(* CODESYS project plc_chalet_xplanar.library
   Title: CHALET_XPlanar
   Version: 5.1.2
   Placeholder: CHALET_XPlanar
   Company: Beckhoff CH

Project tree, tasks and I/O mapping:
  libraries: CHALET_BaseComponents, * (Beckhoff CH); CHALET_Nc, * (Beckhoff CH); Tc2_EtherCAT, * (Beckhoff Automation GmbH); Tc2_Math, * (Beckhoff Automation GmbH); Tc2_Standard, * (Beckhoff Automation GmbH); Tc2_System, * (Beckhoff Automation GmbH); Tc2_Utilities, * (Beckhoff Automation GmbH); Tc3_EventLogger, * (Beckhoff Automation GmbH); Tc3_Mc3Definitions, * (Beckhoff Automation GmbH); Tc3_Mc3PlanarMotion, * (Beckhoff Automation GmbH); Tc3_Module, * (Beckhoff Automation GmbH); Tc3_Physics, * (Beckhoff Automation GmbH); Tc3_XPlanarUtility, * (Beckhoff Automation GmbH)
  COMPONENTs/
    Environment/
      function block FB_XP_Environment [ST]: CollisionCheck, CollisionDetectionAlgorithm, MoverCollisionOffsetError, MoverCollisionOffsetWarning, UpdateCollisionDetection, AddToGroup, RemoveFromGroup, Clear, Configure, FB_init, Feedback, Initialize, Mapped, OID, PlanarEnvironment, Prepare, ProcessingUnitMoverDetectionStatus, ProcessingUnitOID, Update, UtilityEnvirement
      interface I_XP_Enviroment_PLC: CollisionCheck, MoverCollisionOffsetError, MoverCollisionOffsetWarning, MoverDetectionStatus, ProcessingUnitOID
      interface I_XP_Environment: AddToGroup, Clear, Configure, Feedback, Initialize, Mapped, OID, PlanarEnvironment, ProcessingUnitMoverDetectionStatus, ProcessingUnitOID, RemoveFromGroup, Update, UtilityEnvirement
    Feedback/
      function block FB_XP_Feedback [ST]: ClearObjectInfo, ObjectInfo, ObjectInfoEx
      interface I_XP_Feedback: ObjectInfo, ObjectInfoEx
      data type ST_PlanarObjectInfoEx
    Group/
      function block FB_XP_Group [ST]: AddEnvironment, AddMover, AddTrack, Disable, Enable, FB_init, Feedback, Initialize, Mapped, OID, PlanarGroup, Reset, Update
      interface I_XP_Group: AddEnvironment, AddMover, AddTrack, Disable, Enable, Feedback, Initialize, Mapped, OID, PlanarGroup, Reset, Update
    Mover/
      ProductData/
        function block FB_XP_ProductData [ST]: LinkedMover, LinkToMover
        interface I_XP_ProductData: LinkedMover, LinkToMover
      function block FB_XP_Mover [ST]: DynConstraint, SetDynConstraint_A, SetDynConstraint_B, SetDynConstraint_C, SetDynConstraint_Path, SetDynConstraint_X, SetDynConstraint_Y, SetDynConstraint_Z, AddMoverExtSetpoint, AxisExtSetpointA, AxisExtSetpointB, AxisExtSetpointC, AxisExtSetpointX, AxisExtSetpointY, AxisExtSetpointZ, StartExternalSetpoint, StopExternalSetpoint, UpdateExternalSetpoint, AddToGroup, RemoveFromGroup, Halt, MoveA, MoveB, MoveC, MoveXY, MoveZ, Standstill, Disable, Enable, Reset, LastCmdTargedGap, LastCmdTargedPosition, LastCmdTargedTrack, LastValidPositionOnTrack, LastValidPositionXYZABC, LastValidTrack, AccelerationSet, CAxisModulo, CommandMode, DistToParentStation, Enabled, LagDistanceXY, Mapped, Mode, MoverHeight, MoverIsNotPresent, MoverWidth, PositionAct, PositionSet, ProductData, Route, VelocitySet, CurrentTrack, DistToTrack, JoinTrack, MoveOnTrack, MoveOnTrack_ShortestWay, MoveOnTrackToStation, ParentStation, PositionOnTrack, TargetStation, TcIoXPlanarMover, UtilityMover, FB_init, Feedback, Initialize, OID, PlanarMover, Prepare, Update
      interface I_XP_Mover: DynConstraint, SetDynConstraint_A, SetDynConstraint_B, SetDynConstraint_C, SetDynConstraint_Path, SetDynConstraint_X, SetDynConstraint_Y, SetDynConstraint_Z, StopExternalSetpoint, AddToGroup, RemoveFromGroup, Halt, MoveA, MoveB, MoveC, MoveXY, MoveZ, Standstill, Disable, Enable, Reset, LastCmdTargedGap, LastCmdTargedPosition, LastCmdTargedTrack, LastValidPositionOnTrack, LastValidPositionXYZABC, LastValidTrack, AccelerationSet, CAxisModulo, DistToParentStation, Enabled, Feedback, Mapped, Mode, MoverHeight, MoverIsNotPresent, MoverWidth, OID, PositionSet, Route, VelocitySet, CurrentTrack, DistToTrack, JoinTrack, MoveOnTrack, MoveOnTrack_ShortestWay, MoveOnTrackToStation, ParentStation, PositionOnTrack, TargetStation, TcIoXPlanarMover, UtilityMover, PlanarMover
      interface I_XP_Mover_PLC: DynConstraint, SetDynConstraint_A, SetDynConstraint_B, SetDynConstraint_C, SetDynConstraint_Path, SetDynConstraint_X, SetDynConstraint_Y, SetDynConstraint_Z, AxisExtSetpointA, AxisExtSetpointB, AxisExtSetpointC, AxisExtSetpointX, AxisExtSetpointY, AxisExtSetpointZ, StartExternalSetpoint, StopExternalSetpoint, Halt, MoveA, MoveB, MoveC, MoveXY, MoveZ, Standstill, AccelerationSet, CAxisModulo, CommandMode, Enabled, LagDistanceXY, MoverHeight, MoverWidth, PositionAct, PositionSet, VelocitySet, CurrentTrack, LastCmdTargedGap, LastCmdTargedPosition, LastCmdTargedTrack, MoveOnTrack, ParentStation, PositionOnTrack, TargetStation, TcIoXPlanarMover, UtilityMover, DistToParentStation, Feedback, LUID, Mapped, MoverIsNotPresent, OID, PlanarMover, ProductData
    Optional/
      Casting/
        function ToXpMover [ST]
        function ToXpStation [ST]
        function ToXpTrack [ST]
      Trigger/
        function block FB_XP_Trigger [ST]: AccocietedTrack, FB_init, HR, Initialize, ListOfMoversToCheck, MoverAtTrigger, MoverDetected, PositionOnTrack, Prepare, TimeStamp, TriggerDirection, Update
        interface I_XP_Trigger: AccocietedTrack, HR, ListOfMoversToCheck, MoverAtTrigger, MoverDetected, PositionOnTrack, TimeStamp, TriggerDirection
      Zone/
        function block FB_XP_SoretedListOfMover [ST]: CtsMoversInZone, FB_init, Initialize, MoversInZone, Prepare, Update
        interface I_XP_Zone: CtsMoversInZone, MoversInZone
    Path/
      function block FB_XP_Path [ST]: DistanceToDestiantion, Length, LUID, PointerToThis, StationDestination, StationStart, TracksUsed
      interface I_XP_Path: DistanceToDestiantion, Length, PointerToThis, StationDestination, StationStart, TracksUsed
    Stationen/
      A-Star-Node/
        function block FB_AStarNode [ST]: LUID, PathLength, RouteUsedToNode, SortOrderInList, Station
        interface I_PathAStarNode: PathLength, RouteUsedToNode, Station
      function block FB_XP_Station [ST]: CheckInvalideParameter, GetAccocietedTrack, GetDecisionDistance, GetPathsAhead, GetPathsBehind, GetPosOnTrack, GetStationAhead, GetStationBehinde, SetTrackObjName, Configure, CtsEmptySpaceInQueue, CtsMoversInQueue, MoverAccAtExit, MoverDecAtExit, MoverQueueSize, MoversInPlace, MoversInQueue, MoverVelocityAtExit, OnMoverPasses, PushMoversOutOfStation, ReadyToRecvMovers, SendMoversToStation, SuppressDynamicsChange, System, TargetGroupe, TargetPosMonitoringTime, TargetPosWindow, ProcessSimulationActive, SimulationStart, SimulationStartEx, SimulationStop, UpdateSimulation, AccocietedTrack, AddMoverToQueue, AssignedMovers, DeleteMoversQueue, FB_exit, FB_init, Feedback, Filter, GetPathToTarged, Initialize, MoverGapAtExit, OID, PathsAhead, PathsBehinde, PositionOnTrack, PositionOnTrackXY, PositionXY, Prepare, StationsAhead, StationsBehinde, Update, UpdateMoverInteraction
      interface I_XP_Station: AccocietedTrack, AddMoverToQueue, AssignedMovers, Configure, CtsEmptySpaceInQueue, CtsMoversInQueue, DeleteMoversQueue, Filter, MoverAccAtExit, MoverDecAtExit, MoverGapAtExit, MoverQueueSize, MoversInPlace, MoverVelocityAtExit, PathsAhead, PathsBehinde, PositionOnTrack, PositionOnTrackXY, PositionXY, PushMoversOutOfStation, ReadyToRecvMovers, SendMoversToStation, StationsAhead, StationsBehinde, TargetGroupe, Update
      interface I_XP_Station_PLC: CtsEmptySpaceInQueue, CtsMoversInQueue, Filter, LUID, MoverAccAtExit, MoverDecAtExit, MoverQueueSize, MoversInPlace, MoversInQueue, MoverVelocityAtExit, PushMoversOutOfStation, ReadyToRecvMovers, SendMoversToStation, SuppressDynamicsChange, System, TargetPosMonitoringTime, TargetPosWindow, ProcessSimulationActive, SimulationStart, SimulationStartEx, SimulationStop, AccocietedTrack, Feedback, MoverGapAtExit, PositionOnTrack, PositionOnTrackXY, PositionXY, StationsAhead, StationsBehinde, TargetGroupe
    System/
      function block FB_XP_System [ST]: JoiningStation, JoiningTrack, Disable, Disabled, Disabling, Enable, Enabled, Enabling, FastStop, Initialize, Initialized, CheckTargetExists, GetStationClosestTo, Station, LinkEnvironment, LinkGroup, RegisterMover, RegisterStation, RegisterTrack, RegisterTrigger, RegisterZone, CheckForErrors, Enviroment, FB_init, Feedback, Movers, Paths, Stations, SuppressAllDynamicsChanges, Tracks, Triggers, Update, Zones
      interface I_XP_System_PLC: CheckTargetExists, Disable, Disabled, Enable, Enabled, Enviroment, FastStop, Feedback, GetStationClosestTo, Initialize, Initialized, Movers, Paths, Station, Stations, SuppressAllDynamicsChanges, Tracks, Triggers, Update, Zones
      interface I_XP_System_Registration: LinkEnvironment, LinkGroup, RegisterMover, RegisterStation, RegisterTrack, RegisterTrigger, RegisterZone, Disabled, Enabled, Enviroment, Movers, Paths, Stations, Tracks, Triggers, Zones
    Track/
      function block FB_XP_Track [ST]: Configure, Configuring, Disable, Enable, AddToGroup, RemoveFromGroup, AddMover, ClosedLoop, CtsMoversOnTrack, FB_init, Feedback, GapAtPosition, Initialize, Length, Mapped, MoversOnTrack, OID, PathsOnTrack, PlanarTrack, Prepare, Reset, StationAhedPosition, StationsOnTrack, TracksAhead, TracksBehinde, TracksEndAtThis, TracksStartFromThis, Update
      interface I_XP_Track: AddMover, AddToGroup, ClosedLoop, Configure, Configuring, CtsMoversOnTrack, Disable, Enable, Feedback, GapAtPosition, Length, PlanarTrack, RemoveFromGroup, Reset, StationAhedPosition, StationsOnTrack, TracksAhead, TracksBehinde, TracksEndAtThis, TracksStartFromThis
      interface I_XP_Track_PLC: CtsMoversOnTrack, Feedback, Length, Mapped, OID, PlanarTrack, StationAhedPosition, StationsOnTrack, TracksAhead, TracksBehinde, TracksEndAtThis, TracksStartFromThis
  FUNCTIONs/
    function F_DistXYVectors [ST]
    function F_Vector_Multiplication [ST]
    function F_Vector_Subtraction [ST]
    function F_GetDistToPosModulo [ST]
    function F_InLimitTest [ST]
    function F_RotatePositionXY [ST]
    function F_Vector_Addition [ST]
  00000000-0000-0000-0000-000000000000|LICENSE.md
  LICENSE.md
  global variables XPlanarParameterlist
*)

// COMPONENTs/Feedback/ST_PlanarObjectInfoEx
TYPE ST_PlanarObjectInfoEx EXTENDS Tc3_Mc3PlanarMotion.PlanarObjectInfo :
STRUCT
	ipObject : I_CH_Object;
END_STRUCT
END_TYPE

// XPlanarParameterlist
{attribute 'qualified_only'}
VAR_GLOBAL CONSTANT 
	(*After the system init, this is the first station that is approached.
	 Can be used, for example, to send all movers to the “Unload” station first 
	 The default value is “not defined” so the movers remain in the closest station and wait for a valid destination*)
	S_MOVER_TARGED_INIT : STRING := 'not defined';	
	
	(*This value as a Station.Filter allows all movers of any targed*)
	S_ANY_STATION_NAME : STRING := '';
	
	(*Only if enabled, mover take over "VelocytiAtExit" of passed station*)	
	B_STATIONS_OVERRIDE_MOVER_DYN_CONSTRAINT : BOOL := FALSE;

	(*Minimum gap center to center on track [mm] *)
	F_MOVER_MINIMUM_GAP_ON_TRACK : LREAL := 100.0;
	
	(*Default gap center to center on track. Each station can override this gap[mm] *)
	F_GAP_DEFAULT: LREAL := 120.0;
	
	(*Determine the absolute C-rotation of the mover when starting up. Requires an “APM9001-0000-4xxx | XPlanar-ID-Bumper”. *)
	B_GET_MOVER_ORIENTATION : BOOL := FALSE;	
	
	(*Add envirement to groupe during enabling *)
	B_ADD_ENVIROMENT_TO_GROUP : BOOL := TRUE;	
					
	(*Add tracks to groupe during enabling *)
	B_ADD_TRACKS_TO_GROUP : BOOL := FALSE;	
					
	(*Add movers to groupe during enabling *)
	B_ADD_MOVERS_TO_GROUP : BOOL := FALSE;	
					
	(*The movers are only sent to the next free station on the way to the destination. 
	The distance in mm can be specified here to indicate how much further away the new move command can already be sent.  *)
	F_DIST_SET_NEW_MOVE_CMD_BEFORE_REACHING_PARENT_STATION : LREAL := 200.0;
	
	(*max tracks after a track switch *)
	N_MAX_STATIONS_AHEAD_OR_BEHIND : UINT := 20;	
	
	//Velocity during enabling move on track. 0=Default
	F_ENABLING_ON_TRACK_VELOCITY	: LREAL := 0;
	
	//Acc-/Deceleration during enabling move on track. 0=Default
	F_ENABLING_ON_TRACK_ACC_DEC		: LREAL := 0;
	
	//TRUE = Use inside PLC the track name from the TcCom Track Object. If FALSE overwride TcCom Track object with instance name
	B_TRACK_NAME_TACKOVER_FROM_TRACK_OBJECT : BOOL := TRUE;
	

END_VAR

// COMPONENTs/Environment/FB_XP_Environment
{attribute 'no_explicit_call' := 'Do not call the body - Stick to OOP'}
(* XPlanar Environment - 1 per associated XPlanar 
	The Planar environment is a software object that represents the two-dimensional XPlanar stator surface. Together with Planar movers in a group, 
	it prevents collisions of the movers with the edge of the surface. *)
FUNCTION_BLOCK FB_XP_Environment EXTENDS FB_CH_Object IMPLEMENTS I_XP_Environment
VAR
	//Link to Planar-Environment object
	fbEnvironment : MC_PlanarEnvironment;
	fbUtilityEnvirement : FB_TcIoXPlanarEnvironment;
	
	{attribute 'hide'}  
	bInitDone :BOOL := FALSE;
	{attribute 'hide'}
	ipXpSystem : I_XP_System_Registration;
	{attribute 'hide'}               	
	fbFeedback 			: FB_XP_Feedback(ipSourceInfo := fbSourceInfo);	
	{attribute 'hide'}                   	
	eActiveCommand 		: CHALET_Nc.E_NcAxisCommands := CHALET_Nc.E_NcAxisCommands.None;
	{attribute 'hide'}
	bCollisionCheckEnabled : BOOL := TRUE;
	{attribute 'hide'}
	fMoverOffsetWarning : LREAL := 2.0; //[mm]
	{attribute 'hide'}
	fMoverOffsetError: LREAL := 0.0;//[mm]
	{attribute 'hide'}
	eMoverDetectionStatus : MoverDetectionStatus;
	{attribute 'hide'}
	eMoverDetectionStatusLastCycle : MoverDetectionStatus;
END_VAR


// Planar-Feedback objects
VAR
	{attribute 'hide'} 
	fbFeedbackAddToGrp : MC_PlanarFeedback;
	{attribute 'hide'} 
	fbFeedbackRmvFromGrp : MC_PlanarFeedback;
	{attribute 'hide'} 
	fbFeedbackConfigure : MC_PlanarFeedback;
	{attribute 'hide'} 
	fbFeedbackClear : MC_PlanarFeedback;
END_VAR

{attribute 'monitoring':='call'}
(* If Enable, the movers are checked for collisions with each other.
Warning and error can have their own size offsets.
The error leads to a stop with higher dynamics.
In simulation, an error does not lead to a stop *)
PROPERTY CollisionCheck : BOOL
GET
CollisionCheck := THIS^.bCollisionCheckEnabled;
END_GET
SET
THIS^.bCollisionCheckEnabled := CollisionCheck;
END_SET
END_PROPERTY

//Return an interface to the mover if a collision is active else return 0. The check stops after the first collision found
METHOD PROTECTED CollisionDetectionAlgorithm : I_XP_Mover
VAR_INPUT
	ipListOfMovers : I_CH_LIST;
	fOffsetMoverSize : LREAL := 1.0; //Offset on the mover dimension from the MC3 mover object [mm];
END_VAR
VAR
	aPointsMover1 : ARRAY[0..3] OF  Tc3_Physics.PositionXY;
	aPointsEachMover : ARRAY[0..3] OF  Tc3_Physics.PositionXY;
	aPointsDelta : ARRAY[0..3] OF  Tc3_Physics.PositionXY;
	
	fMoverWidth, fMoverHight : LREAL;
	fMoverXPos, fMoverYPos, fMoverCPos : LREAL;
	
	ipMover1, ipEachMover : I_XP_Mover;
	fbListOfMoverToCheck : FB_CH_List;
	
	fAngle : LREAL;
	a, b, c: LREAL;
	Pa, Pb, Pc : REFERENCE TO Tc3_Physics.PositionXY;
	fcos : LREAL;
	
	nIdx, nIdxMover1, nIdxPlus1 : UINT;
	ipMover2CollisionFound : I_XP_Mover;
END_VAR
//Get all mover in a list
fbListOfMoverToCheck.Duplicate(ipListOfMovers);



//Check list for invalide Act Pos - ex.: if mover is not found 
fbListOfMoverToCheck.ResetIterator();
WHILE fbListOfMoverToCheck.HasNextObject() DO
	__QUERYINTERFACE(fbListOfMoverToCheck.GetNextObject(),ipMover1);
	
	IF ipMover1.MoverIsNotPresent THEN 		
		//remove from list
		fbListOfMoverToCheck.RemoveObject(ipMover1);
		
	END_IF
END_WHILE



fbListOfMoverToCheck.ResetIterator();
WHILE fbListOfMoverToCheck.HasNextObject() DO
	//get first mover in list,
	__QUERYINTERFACE(fbListOfMoverToCheck.GetNextObject(),ipMover1);
	
	fMoverXPos := ipMover1.PlanarMover.MCTOPLC.ACT.ActPos.x;
	fMoverYPos := ipMover1.PlanarMover.MCTOPLC.ACT.ActPos.y;
	fMoverCPos := ipMover1.PlanarMover.MCTOPLC.ACT.ActPos.c;
		
	//Get corner points of the rectangle 
	fMoverWidth := ipMover1.MoverWidth - fOffsetMoverSize;
	fMoverHight := ipMover1.MoverHeight - fOffsetMoverSize;
	aPointsMover1[0].SetValuesXY(x:= -fMoverWidth/2, y:= -fMoverHight/2);//Bottom Left
	aPointsMover1[1].SetValuesXY(x:= -fMoverWidth/2, y:=  fMoverHight/2);//Top Left
	aPointsMover1[2].SetValuesXY(x:=  fMoverWidth/2, y:=  fMoverHight/2);//Top Ritgh
	aPointsMover1[3].SetValuesXY(x:=  fMoverWidth/2, y:= -fMoverHight/2);//Bottom Rigth
	
	//Rotation of the mover
	F_RotatePositionXY(aPointsMover1[0], fMoverCPos);
	F_RotatePositionXY(aPointsMover1[1], fMoverCPos);
	F_RotatePositionXY(aPointsMover1[2], fMoverCPos);
	F_RotatePositionXY(aPointsMover1[3], fMoverCPos);
	
	//shift to mover coordinates
	aPointsMover1[0].ShiftByXY(dx:= fMoverXPos, dy:= fMoverYPos);
	aPointsMover1[1].ShiftByXY(dx:= fMoverXPos, dy:= fMoverYPos);
	aPointsMover1[2].ShiftByXY(dx:= fMoverXPos, dy:= fMoverYPos);
	aPointsMover1[3].ShiftByXY(dx:= fMoverXPos, dy:= fMoverYPos);
	
	
	//do an check for all mover
	fbListOfMoverToCheck.ResetIterator();
	WHILE fbListOfMoverToCheck.HasNextObject() DO
		__QUERYINTERFACE(fbListOfMoverToCheck.GetNextObject(),ipEachMover);
		
		IF ipEachMover = ipMover1 THEN
			//Skip if same
			CONTINUE;
		END_IF
		
		fMoverXPos := ipEachMover.PlanarMover.MCTOPLC.ACT.ActPos.x;
		fMoverYPos := ipEachMover.PlanarMover.MCTOPLC.ACT.ActPos.y;
		fMovercPos := ipEachMover.PlanarMover.MCTOPLC.ACT.ActPos.c;
		
		//Get corner points of the rectangle 
		fMoverWidth := ipEachMover.MoverWidth - fOffsetMoverSize;
		fMoverHight := ipEachMover.MoverHeight - fOffsetMoverSize;
		aPointsEachMover[0].SetValuesXY(x:= -fMoverWidth/2, y:= -fMoverHight/2);//Bottom Left
		aPointsEachMover[1].SetValuesXY(x:= -fMoverWidth/2, y:=  fMoverHight/2);//Top Left
		aPointsEachMover[2].SetValuesXY(x:=  fMoverWidth/2, y:=  fMoverHight/2);//Top Ritgh
		aPointsEachMover[3].SetValuesXY(x:=  fMoverWidth/2, y:= -fMoverHight/2);//Bottom Rigth

		//Rotation of the mover
		F_RotatePositionXY(aPointsEachMover[0], fMoverCPos);
		F_RotatePositionXY(aPointsEachMover[1], fMoverCPos);
		F_RotatePositionXY(aPointsEachMover[2], fMoverCPos);
		F_RotatePositionXY(aPointsEachMover[3], fMoverCPos);
		
		//shift to mover coordinates
		aPointsEachMover[0].ShiftByXY(dx:= fMoverXPos, dy:= fMoverYPos);
		aPointsEachMover[1].ShiftByXY(dx:= fMoverXPos, dy:= fMoverYPos);
		aPointsEachMover[2].ShiftByXY(dx:= fMoverXPos, dy:= fMoverYPos);
		aPointsEachMover[3].ShiftByXY(dx:= fMoverXPos, dy:= fMoverYPos);		
		
		//check each corener if inside each mover
		FOR nIdxMover1 := 0 TO 3 DO
			
			(* A triangle is created between a corner point of Mover1 (point a) and two corner points of Mover2 (points B and C). 
			All corner points of Mover2 are now tested one after the other. If the sum of all angles "a" is 360 degrees, 
			then point A is inside mover 2 and there is a collision *)
			fAngle := 0;
			FOR nIdx := 0 TO 3 DO
				nIdxPlus1 := ((nIdx+1)MOD 4);
			
				Pa REF= aPointsMover1[nIdxMover1];
				Pb REF= aPointsEachMover[nIdx];
				Pc REF= aPointsEachMover[nIdxPlus1];					
				

				a := SQRT(EXPT((Pb.x - Pc.x),2)+EXPT((Pb.y - Pc.y),2));
				b := SQRT(EXPT((Pa.x - Pc.x),2)+EXPT((Pa.y - Pc.y),2));
				c := SQRT(EXPT((Pa.x - Pb.x),2)+EXPT((Pa.y - Pb.y),2));
				
				
				IF b=0 OR c=0 THEN
					//Error - Return the found mover
					CollisionDetectionAlgorithm := ipMover1;
					//with which mover is the collision
					ipMover2CollisionFound := ipEachMover;
					RETURN;
				ELSE
					(*  a/sin(α) = b/sin(β) = c/sin(γ) *)
					fcos := (EXPT(b,2) + EXPT(c,2) - EXPT(a,2))/(2*b*c);
					fcos := LIMIT(-1.0, fcos, 1.0);
					fAngle :=  fAngle + ACOS(fcos);
				END_IF
			END_FOR
			
			//if the point is inside the mover, the sum of all angles is exactly 360°-> 2pi
			IF ABS(fAngle - 2*Tc2_System.PI)<0.01 THEN
				//Error - Return the found mover
				CollisionDetectionAlgorithm := ipMover1;
				//with which mover is the collision
				ipMover2CollisionFound := ipEachMover;
				RETURN;
			END_IF
			
		END_FOR

	END_WHILE
	fbListOfMoverToCheck.RestoreIterator();
	
	
	
END_WHILE
END_METHOD

{attribute 'monitoring':='call'}
//Offset on the mover dimension from the MC3 mover object [mm] ;
// >0 menas the warning is earlier
PROPERTY MoverCollisionOffsetError : LREAL
GET
MoverCollisionOffsetError := fMoverOffsetError;
END_GET
SET
fMoverOffsetError := MoverCollisionOffsetError;
END_SET
END_PROPERTY

{attribute 'monitoring':='call'}
//Offset on the mover dimension from the MC3 mover object [mm] ;
// >0 menas the warning is earlier
PROPERTY MoverCollisionOffsetWarning : LREAL
GET
MoverCollisionOffsetWarning :=  fMoverOffsetWarning;
END_GET
SET
fMoverOffsetWarning := MoverCollisionOffsetWarning;
END_SET
END_PROPERTY

METHOD PROTECTED UpdateCollisionDetection : HRESULT
VAR
	bDisableDuringMoverDetection : BOOL;
	ipMoverCollision : I_XP_Mover;
	ipSystemPlc : I_XP_System_PLC;
	nX, nY : DINT;
END_VAR
VAR_INST
	{attribute 'hide'}	
	ipMoverCollisionOldWarning : I_XP_Mover;
	{attribute 'hide'}	
	fbAlarmCollisionMoverWarning : FB_TcAlarm;	
	{attribute 'hide'}	
	ipMoverCollisionOldAlarm : I_XP_Mover;
	{attribute 'hide'}	
	fbAlarmCollisionMoverAlarm : FB_TcAlarm;
END_VAR
bDisableDuringMoverDetection := THIS^.ProcessingUnitMoverDetectionStatus = MoverDetectionStatus.DetectionInProcess;


//Check whether a mover has a collision with another mover and generate a warning.
//Only 1 mover is found and displayed
//WARNING - each mover default is 2mm larger
IF THIS^.bCollisionCheckEnabled AND NOT bDisableDuringMoverDetection THEN
	//get mover or 0 for no collision
	ipMoverCollision := CollisionDetectionAlgorithm(fOffsetMoverSize := THIS^.fMoverOffsetWarning, ipListOfMovers := THIS^.ipXpSystem.Movers);
	
	IF ipMoverCollision <> 0 AND_THEN ipMoverCollision <> ipMoverCollisionOldWarning AND_THEN NOT ipMoverCollision.MoverIsNotPresent THEN
		fbAlarmCollisionMoverWarning.CreateEx(tc_Events.CHALET_XPlanar_Events.MoverCollisionWarning, 0, THIS^.fbSourceInfo);
		//Mover "{0}" has a collision with another mover at position X:{1} Y:{2}
		nX := LREAL_TO_DINT(ipMoverCollision.PlanarMover.MCTOPLC.ACT.ActPos.x);
		nY := LREAL_TO_DINT(ipMoverCollision.PlanarMover.MCTOPLC.ACT.ActPos.y);
		fbAlarmCollisionMoverWarning.ipArguments.Clear().AddStringByValue(ipMoverCollision.LUID).AddDInt(nX).AddDint(nY);
		fbAlarmCollisionMoverWarning.Raise(0);
	ELSIF ipMoverCollision = 0 THEN
		//No collision found
		fbAlarmCollisionMoverWarning.Clear(0,0);
	END_IF
	ipMoverCollisionOldWarning := ipMoverCollision;
ELSE
	fbAlarmCollisionMoverWarning.Clear(0,0);
	ipMoverCollisionOldWarning := 0;
END_IF

//Check whether a mover has a collision with another mover and generate a warning.
//Only 1 mover is found and displayed
//ERROR - each mover is default -1mm smaller
IF THIS^.bCollisionCheckEnabled AND NOT bDisableDuringMoverDetection  THEN
	//get mover or 0 for no collision
	ipMoverCollision := CollisionDetectionAlgorithm(fOffsetMoverSize := THIS^.fMoverOffsetError, ipListOfMovers := THIS^.ipXpSystem.Movers);
	
	IF ipMoverCollision <> 0 AND ipMoverCollision <> ipMoverCollisionOldAlarm THEN
		fbAlarmCollisionMoverAlarm.CreateEx(tc_Events.CHALET_XPlanar_Events.MoverCollisionStop, 0, THIS^.fbSourceInfo);
		//Mover "{0}" has a collision with another mover at position X:{1} Y:{2}
		fbAlarmCollisionMoverAlarm.ipArguments.AddStringByValue(ipMoverCollision.LUID).AddUDInt(LREAL_TO_UDINT(ipMoverCollision.PlanarMover.MCTOPLC.ACT.ActPos.x)).AddUDInt(LREAL_TO_UDINT(ipMoverCollision.PlanarMover.MCTOPLC.ACT.ActPos.y));
		fbAlarmCollisionMoverAlarm.Raise(0);

		//Stop if this is a real system, keep running in simulation
		IF THIS^.UtilityEnvirement.XpuTcIo(1).GetOperationMode() = OperationMode.Normal THEN
			IF __QUERYINTERFACE(THIS^.ipXpSystem, ipSystemPlc) THEN
				//Disable System
				ipSystemPlc.FastStop();
			END_IF
		END_IF
	ELSIF ipMoverCollision = 0 THEN
		//No collision found
		fbAlarmCollisionMoverAlarm.Clear(0,0);
	END_IF
		
	ipMoverCollisionOldAlarm := ipMoverCollision;
ELSE
	fbAlarmCollisionMoverAlarm.Clear(0,0);
	ipMoverCollisionOldAlarm := 0;
END_IF
END_METHOD

METHOD AddToGroup : HRESULT
VAR_INPUT
	iGroup : I_XP_Group;
END_VAR
IF NOT THIS^.fbFeedback.Busy THEN
	THIS^.eActiveCommand 				:= CHALET_NC.E_NcAxisCommands.AddToGroupe;
	THIS^.fbFeedback.LastCommandAccepted:= TRUE;		
	THIS^.fbFeedback.Busy 				:= TRUE;
	
	iGroup.AddEnvironment(THIS^.fbEnvironment, THIS^.fbFeedbackAddToGrp);
	AddToGroup := S_OK;
ELSE
	AddToGroup := S_FALSE;
	THIS^.fbFeedback.LastCommandAccepted:= FALSE;	
END_IF
END_METHOD

METHOD RemoveFromGroup : HRESULT
IF NOT THIS^.fbFeedback.Busy THEN
	THIS^.eActiveCommand 				:= CHALET_NC.E_NcAxisCommands.RemoveFromGroupe;
	THIS^.fbFeedback.LastCommandAccepted:= TRUE;		
	THIS^.fbFeedback.Busy 				:= TRUE;
	
	THIS^.fbEnvironment.RemoveFromGroup(THIS^.fbFeedbackRmvFromGrp);
	RemoveFromGroup := S_OK;
ELSE
	RemoveFromGroup := S_FALSE;
	THIS^.fbFeedback.LastCommandAccepted:= FALSE;	
END_IF
END_METHOD

METHOD Clear : HRESULT
THIS^.eActiveCommand 				:= CHALET_NC.E_NcAxisCommands.Clear;
THIS^.fbFeedback.LastCommandAccepted:= TRUE;		
THIS^.fbFeedback.Busy 				:= TRUE;

THIS^.fbEnvironment.Clear(commandFeedback:=THIS^.fbFeedbackClear);
Clear := S_OK;
END_METHOD

METHOD Configure : HRESULT
THIS^.eActiveCommand 				:= CHALET_NC.E_NcAxisCommands.Configure;
THIS^.fbFeedback.LastCommandAccepted:= TRUE;		
THIS^.fbFeedback.Busy 				:= TRUE;

THIS^.fbEnvironment.CreateBoundary(commandFeedback:=THIS^.fbFeedbackConfigure);
Configure := S_OK;
END_METHOD

METHOD FB_init : BOOL
VAR_INPUT
	bInitRetains : BOOL; // if TRUE, the retain variables are initialized (warm start / cold start)
	bInCopyCode : BOOL;  // if TRUE, the instance afterwards gets moved into the copy code (online change)
	
	ipSystem : I_CH_Object;
END_VAR
VAR_INST
	{attribute 'hide'}
	bFBInitCalledOnce : BOOL; //Do the following code once during start up and not during onlinechange
END_VAR
//Do the following code once during start up and not during onlinechange
IF NOT bFBInitCalledOnce THEN 
	
	(* Register to the Xplanar System
	   1. Test if the interface exists
	   2. Test if the object implements a "System for Mover" interface 
	*)
	IF ipSystem <> 0 AND_THEN __QUERYINTERFACE(ipSystem,THIS^.ipXpSystem) THEN
		THIS^.ipXpSystem.LinkEnvironment(THIS^);
	END_IF
	
	
END_IF

bFBInitCalledOnce := TRUE;
END_METHOD

{attribute 'monitoring':='call'}
PROPERTY Feedback : I_XP_Feedback
GET
Feedback := THIS^.fbFeedback;
END_GET
END_PROPERTY

METHOD Initialize : HRESULT
VAR
	stVarInfo : __SYSTEM.VAR_INFO;
END_VAR
VAR_INST
	//This error cannot be reset. Requires a reset cold
	{attribute 'hide'}	
	fbInitError : FB_TcAlarm;
END_VAR
// Check if link to envirement is mapped
IF NOT THIS^.Mapped THEN
	IF NOT fbInitError.bRaised THEN 
		//This error cannot be reset. Requires a reset cold
		fbInitError.CreateEx(stEventEntry:=TC_EVENTS.CHALET_Base_Events.VariableLinkMissing, ipSourceInfo := THIS^.fbSourceInfo, bWithConfirmation := FALSE);
		stVarInfo := __VARINFO(fbEnvironment);
		fbInitError.ipArguments.AddString(stVarInfo.Symbol);
		fbInitError.Raise(0);
	END_IF
	Initialize := E_FAIL;
	RETURN;
END_IF



IF NOT bInitDone THEN
	//Busy
	Initialize := S_PENDING;
	
	IF fbUtilityEnvirement.Init(bExecute := TRUE) THEN
		fbUtilityEnvirement.Init(bExecute := FALSE);
		bInitDone := TRUE;
	END_IF
	
	
ELSE	
	//Done
	Initialize := S_OK;
END_IF



THIS^.fbFeedback.ActiveCommand 		:= TO_STRING(CHALET_NC.E_NcAxisCommands.Initialize);
THIS^.eActiveCommand 				:= CHALET_NC.E_NcAxisCommands.Initialize;
THIS^.fbFeedback.LastCommandAccepted:= TRUE;	
//Set done or keep in busy state	
THIS^.fbFeedback.HR := Initialize;
END_METHOD

{attribute 'monitoring':='call'}
PROPERTY Mapped : BOOL //Project is mapped to MC (McToPlc and PlcToMc)
GET
VAR
	bMcToPlcNotMapped 	: BOOL;
END_VAR
bMcToPlcNotMapped := F_GetMappingStatus(ADR(THIS^.fbEnvironment.MCTOPLC_STD), SIZEOF(THIS^.fbEnvironment.MCTOPLC_STD)) <> EPlcMappingStatus.MS_Mapped;

Mapped := NOT bMcToPlcNotMapped;
END_GET
END_PROPERTY

{attribute 'monitoring':='call'}
//Unique object ID
PROPERTY OID : OTCID
GET
OID := THIS^.fbEnvironment.MCTOPLC_STD.EnvironmentOID;
END_GET
END_PROPERTY

{attribute 'monitoring':='call'}
PROPERTY PlanarEnvironment : REFERENCE TO MC_PlanarEnvironment
GET
PlanarEnvironment ref= THIS^.fbEnvironment;
END_GET
END_PROPERTY

(* Time-critical information is processed here, which can then be polled via the property every cycle. 
The update method is usually at the end of the program and then it is already 'outdated'. *)
METHOD PRIVATE Prepare : HRESULT
VAR CONSTANT
	N_IDX_OFFSET_MoverDetectionStatus 	: UDINT := 16#03171005; // Parameter(online) in Planar  Processing Unit object 
END_VAR
VAR
	nParaSize : UDINT;
	pParaData : PVOID;
	hr : HRESULT;
	ipComObject : ITComObject;
END_VAR
VAR_INST
	{attribute 'hide'}
	nLastUpdatedCycleCount : UDINT;
END_VAR
//Check if this Cycle the dates are allready prepared
IF nLastUpdatedCycleCount <> TwinCAT_SystemInfoVarList._TaskInfo[THIS^.nTaskIndex].CycleCount THEN
	nLastUpdatedCycleCount := TwinCAT_SystemInfoVarList._TaskInfo[THIS^.nTaskIndex].CycleCount;

	
	//************** Read MoverDetectionStatus **************
	//Get interface to ComObject
	FW_ObjMgr_GetObjectInstance(oid:= THIS^.ProcessingUnitOID, iid:= TC_GLOBAL_IID_LIST.IID_ITComObject, pipUnk:= ADR(ipComObject));
	
	//Get ADR and SIZE
	nParaSize := SIZEOF(eMoverDetectionStatus);	pParaData := ADR(eMoverDetectionStatus);
	
	IF ipComObject <> 0 THEN
		hr := ipComObject.TcGetObjPara(pid:=N_IDX_OFFSET_MoverDetectionStatus , nData:= nParaSize, pData:= pParaData, pgp:=0 );	
		ipComObject.TcRelease();	
	END_IF
	
	//force to have the in progress active FOR 1 cycle longer
	IF eMoverDetectionStatus = MoverDetectionStatus.DetectionSuccessful AND eMoverDetectionStatusLastCycle = MoverDetectionStatus.DetectionInProcess THEN
		//Store info from last cycle
		eMoverDetectionStatusLastCycle := eMoverDetectionStatus;
		eMoverDetectionStatus := MoverDetectionStatus.DetectionInProcess;
	ELSE	
		//Store info from last cycle
		eMoverDetectionStatusLastCycle := eMoverDetectionStatus;
	END_IF
	


		
END_IF
END_METHOD

{attribute 'monitoring':='call'}
//Enumeration MoverDetectionStatus
PROPERTY ProcessingUnitMoverDetectionStatus : MoverDetectionStatus
GET
THIS^.Prepare();//Prepare time-critical information, if not already done


ProcessingUnitMoverDetectionStatus := THIS^.eMoverDetectionStatus;
END_GET
END_PROPERTY

{attribute 'monitoring':='call'}
//Object ID of the IoXPlanar processing unit
PROPERTY ProcessingUnitOID : OTCID
GET
VAR
	nProcessingUnitOid : OTCID;
END_VAR
VAR CONSTANT
	N_IDX_OFFSET_PU_Oid 	: UDINT := 16#050300C0; // Parameter(online) in Planar Environment object 
END_VAR

VAR
	nParaSize : UDINT;
	pParaData : PVOID;
	hr : HRESULT;
	ipComObject : ITComObject;
	nOid : OTCID;
END_VAR
//Get TcCom Object ID
nOid := THIS^.OID;

//Get interface to ComObject
FW_ObjMgr_GetObjectInstance(oid:= nOid, iid:= TC_GLOBAL_IID_LIST.IID_ITComObject, pipUnk:= ADR(ipComObject));

//Get ADR and SIZE
nParaSize := SIZEOF(nProcessingUnitOid);	pParaData := ADR(nProcessingUnitOid);

IF ipComObject <> 0 THEN
	hr := ipComObject.TcGetObjPara(pid:=N_IDX_OFFSET_PU_Oid , nData:= nParaSize, pData:= pParaData, pgp:=0 );	
	ipComObject.TcRelease();	
END_IF

ProcessingUnitOID := nProcessingUnitOid;
END_GET
END_PROPERTY

METHOD PUBLIC Update : HRESULT



// ********************** Set feedback depending on active command *******************************
IF THIS^.eActiveCommand <> E_NcAxisCommands.None THEN
	fbFeedback.ActiveCommand 	:= TO_STRING(THIS^.eActiveCommand);	
END_IF

CASE THIS^.eActiveCommand OF
	E_NcAxisCommands.None: 
		//Display if a Mover Error is active during no command is active
		IF THIS^.fbEnvironment.Error AND NOT fbFeedback.Error THEN 
			fbFeedback.ErrorId 			:= THIS^.fbEnvironment.ErrorID;
			fbFeedback.ActiveCommand 	:= TO_STRING(E_NcAxisCommands.None);	
			fbFeedback.ClearObjectInfo();
		END_IF

	E_NcAxisCommands.Initialize:
		fbFeedback.Busy 			:= NOT THIS^.bInitDone;
		fbFeedback.Done 			:= THIS^.bInitDone;
		fbFeedback.ErrorId 			:= 0;
		fbFeedback.ClearObjectInfo();
		                                                       			                        	
	E_NcAxisCommands.Clear:     	
		fbFeedback.Busy 			:= fbFeedbackClear.Busy;
		fbFeedback.Done 			:= fbFeedbackClear.Done;
		fbFeedback.ErrorId 			:= fbFeedbackClear.ErrorID;
        fbFeedback.ObjectInfo		:= fbFeedbackClear.objectInfo;
           			                        	
	E_NcAxisCommands.Configure:     	
		fbFeedback.Busy 			:= fbFeedbackConfigure.Busy;
		fbFeedback.Done 			:= fbFeedbackConfigure.Done;
		fbFeedback.ErrorId 			:= fbFeedbackConfigure.ErrorID;
        fbFeedback.ObjectInfo		:= fbFeedbackConfigure.objectInfo;
                                      			                        	
	E_NcAxisCommands.AddToGroupe:     	
		fbFeedback.Busy 			:= fbFeedbackAddToGrp.Busy;
		fbFeedback.Done 			:= fbFeedbackAddToGrp.Done;
		fbFeedback.ErrorId 			:= fbFeedbackAddToGrp.ErrorID;
        fbFeedback.ObjectInfo		:= fbFeedbackAddToGrp.objectInfo;
                                      			                        	
	E_NcAxisCommands.RemoveFromGroupe:     	
		fbFeedback.Busy 			:= fbFeedbackRmvFromGrp.Busy;
		fbFeedback.Done 			:= fbFeedbackRmvFromGrp.Done;
		fbFeedback.ErrorId 			:= fbFeedbackRmvFromGrp.ErrorID;
        fbFeedback.ObjectInfo		:= fbFeedbackRmvFromGrp.objectInfo;
                                		
	ELSE//External command in subclass
		;
END_CASE


// **********************  Stop to execute commands on .done or .error ***************************
IF fbFeedback.Done OR THIS^.fbFeedback.Error THEN
	eActiveCommand 				:= E_NcAxisCommands.None;
END_IF





//Update Collision subroutin
THIS^.UpdateCollisionDetection();


//Update xplanar object
THIS^.fbEnvironment.Update();

//Update feedback object
fbFeedbackConfigure.Update(); 
fbFeedbackClear.Update(); 
fbFeedbackAddToGrp.Update(); 
fbFeedbackRmvFromGrp.Update();
END_METHOD

{attribute 'monitoring':='call'}
PROPERTY UtilityEnvirement : Tc3_XPlanarUtility.I_Environment
GET
UtilityEnvirement := fbUtilityEnvirement;
END_GET
END_PROPERTY

END_FUNCTION_BLOCK

// COMPONENTs/Environment/I_XP_Environment
INTERFACE I_XP_Environment EXTENDS I_CH_Object

METHOD AddToGroup : HRESULT
VAR_INPUT
	iGroup : I_XP_Group;
END_VAR
END_METHOD

METHOD Clear : HRESULT
END_METHOD

METHOD Configure : HRESULT
VAR_INPUT
END_VAR
END_METHOD

{attribute 'monitoring':='call'}
PROPERTY Feedback : I_XP_Feedback
GET
END_GET
END_PROPERTY

METHOD Initialize : HRESULT
END_METHOD

{attribute 'monitoring':='call'}
PROPERTY Mapped : BOOL //Project is mapped to MC (McToPlc and PlcToMc)
GET
END_GET
END_PROPERTY

{attribute 'monitoring':='call'}
//Unique object ID
PROPERTY OID : OTCID
GET
END_GET
END_PROPERTY

{attribute 'monitoring':='call'}
PROPERTY PlanarEnvironment : REFERENCE TO MC_PlanarEnvironment
GET
END_GET
END_PROPERTY

{attribute 'monitoring':='call'}
//Enumeration MoverDetectionStatus
PROPERTY ProcessingUnitMoverDetectionStatus : MoverDetectionStatus
GET
END_GET
END_PROPERTY

{attribute 'monitoring':='call'}
//Object ID of the IoXPlanar processing unit
PROPERTY ProcessingUnitOID : OTCID
GET
END_GET
END_PROPERTY

METHOD RemoveFromGroup : HRESULT
END_METHOD

METHOD PUBLIC Update : HRESULT
VAR_INPUT
END_VAR
END_METHOD

{attribute 'monitoring':='call'}
PROPERTY UtilityEnvirement : Tc3_XPlanarUtility.I_Environment
GET
END_GET
END_PROPERTY

END_INTERFACE

// COMPONENTs/Group/I_XP_Group
INTERFACE I_XP_Group  EXTENDS I_CH_Object

METHOD AddEnvironment : HRESULT
VAR_INPUT
	refEnvironment : REFERENCE TO MC_PlanarEnvironment;
	refFeedback : REFERENCE TO MC_PlanarFeedback;
END_VAR
END_METHOD

METHOD AddMover : HRESULT
VAR_INPUT
	refMover : REFERENCE TO MC_PlanarMover;
	refFeedback : REFERENCE TO MC_PlanarFeedback;
END_VAR
END_METHOD

METHOD AddTrack : HRESULT
VAR_INPUT
	refTrack : REFERENCE TO MC_PlanarTrack;
	refFeedback : REFERENCE TO MC_PlanarFeedback;
END_VAR
END_METHOD

METHOD Disable : HRESULT
VAR_INPUT
END_VAR
END_METHOD

METHOD Enable : HRESULT
VAR_INPUT
END_VAR
END_METHOD

{attribute 'OPC.UA.DA.Property' := '1'}
{attribute 'monitoring':='call'}
PROPERTY Feedback : I_XP_Feedback
GET
END_GET
END_PROPERTY

METHOD Initialize : HRESULT
VAR_INPUT
END_VAR
END_METHOD

{attribute 'monitoring':='call'}
PROPERTY Mapped : BOOL //Project is mapped to MC (McToPlc and PlcToMc)
GET
END_GET
END_PROPERTY

{attribute 'monitoring':='call'}
//Unique object ID
PROPERTY OID : OTCID
GET
END_GET
END_PROPERTY

{attribute 'monitoring':='call'}
PROPERTY PlanarGroup : REFERENCE TO MC_PlanarGroup
GET
END_GET
END_PROPERTY

METHOD Reset : HRESULT
VAR_INPUT
END_VAR
END_METHOD

METHOD PUBLIC Update : HRESULT
VAR_INPUT
END_VAR
END_METHOD

END_INTERFACE

// COMPONENTs/Feedback/I_XP_Feedback
INTERFACE I_XP_Feedback EXTENDS CHALET_BaseComponents.I_CH_Feedback

{attribute 'monitoring':='call'}
(* Indicates which object one would collide with. *)
PROPERTY ObjectInfo : REFERENCE TO PlanarObjectInfo
GET
END_GET
SET
END_SET
END_PROPERTY

{attribute 'monitoring':='call'}
(* Indicates which object one would collide with. *)
PROPERTY ObjectInfoEx : REFERENCE TO ST_PlanarObjectInfoEx
GET
END_GET
SET
END_SET
END_PROPERTY

END_INTERFACE

// COMPONENTs/System/I_XP_System_Registration
INTERFACE I_XP_System_Registration EXTENDS __SYSTEM.IQueryInterface

METHOD LinkEnvironment : HRESULT
VAR_INPUT
	ipEnvironment : I_CH_Object;
END_VAR
END_METHOD

METHOD LinkGroup : HRESULT
VAR_INPUT
	ipGroup : I_CH_Object;
END_VAR
END_METHOD

METHOD RegisterMover : HRESULT
VAR_INPUT
	ipMover : I_CH_Object;
END_VAR
END_METHOD

METHOD RegisterStation : HRESULT
VAR_INPUT
	ipStation : I_CH_Object;
END_VAR
END_METHOD

METHOD RegisterTrack : HRESULT
VAR_INPUT
	ipTrack : I_CH_Object;
END_VAR
END_METHOD

METHOD RegisterTrigger : HRESULT
VAR_INPUT
	ipTrigger	: CHALET_BaseComponents.I_CH_Object;
END_VAR
END_METHOD

METHOD RegisterZone : HRESULT
VAR_INPUT
	ipZone	: CHALET_BaseComponents.I_CH_Object;
END_VAR
END_METHOD

{attribute 'monitoring':='call'}
PROPERTY Disabled : BOOL
GET
END_GET
END_PROPERTY

{attribute 'monitoring':='call'}
PROPERTY Enabled : BOOL
GET
END_GET
END_PROPERTY

{attribute 'monitoring':='call'}
PROPERTY Enviroment : I_XP_Environment
GET
END_GET
END_PROPERTY

{attribute 'monitoring':='call'}
PROPERTY Movers : CHALET_BaseComponents.I_CH_LIST
GET
END_GET
END_PROPERTY

{attribute 'monitoring':='call'}
PROPERTY Paths : CHALET_BaseComponents.I_CH_LIST
GET
END_GET
END_PROPERTY

{attribute 'monitoring':='call'}
PROPERTY Stations : CHALET_BaseComponents.I_CH_LIST
GET
END_GET
END_PROPERTY

{attribute 'monitoring':='call'}
PROPERTY Tracks : CHALET_BaseComponents.I_CH_LIST
GET
END_GET
END_PROPERTY

{attribute 'monitoring':='call'}
PROPERTY Triggers : CHALET_BaseComponents.I_CH_LIST
GET
END_GET
END_PROPERTY

{attribute 'monitoring':='call'}
PROPERTY Zones : CHALET_BaseComponents.I_CH_LIST
GET
END_GET
END_PROPERTY

END_INTERFACE

// COMPONENTs/Feedback/FB_XP_Feedback
{attribute 'no_explicit_call' := 'Do not call the body - Stick to OOP'}
FUNCTION_BLOCK FB_XP_Feedback EXTENDS CHALET_BaseComponents.FB_CH_Feedback IMPLEMENTS I_XP_Feedback
VAR_INPUT
END_VAR
VAR_OUTPUT
END_VAR
VAR
	(* Indicates which object one would collide with. *)
	{attribute 'hide'}
	_objectInfo : ST_PlanarObjectInfoEx;
END_VAR

METHOD ClearObjectInfo : BOOL
VAR_INPUT
END_VAR
THIS^._ObjectInfo.Id := 0;
THIS^._ObjectInfo.ipObject := 0;
THIS^._ObjectInfo.ObjectType := EPlanarObjectType.None;
END_METHOD

{attribute 'monitoring':='call'}
(* Indicates which object one would collide with. *)
PROPERTY ObjectInfo : REFERENCE TO PlanarObjectInfo
GET
objectInfo REF= THIS^._objectInfo;
END_GET
SET
THIS^._objectInfo.Id			:= ObjectInfo.Id;
THIS^._objectInfo.ObjectType 	:= ObjectInfo.ObjectType;
THIS^._objectInfo.ipObject 		:= 0;
END_SET
END_PROPERTY

{attribute 'monitoring':='call'}
(* Indicates which object one would collide with. *)
PROPERTY ObjectInfoEx : REFERENCE TO ST_PlanarObjectInfoEx
GET
objectInfoEx REF= THIS^._objectInfo;
END_GET
SET
THIS^._objectInfo := ObjectInfoEx;
END_SET
END_PROPERTY

END_FUNCTION_BLOCK

// FUNCTIONs/F_RotatePositionXY
//Rotate a point (XY) around its 0-point. 
//e.g. from (10/0)+90°-> (0/10) 
FUNCTION F_RotatePositionXY : HRESULT
VAR_INPUT
	fbPosition : REFERENCE TO Tc3_Physics.PositionXY;
	fRotate : LREAL; //[°]
END_VAR
VAR
	fRadius : LREAL;
	fPhi : LREAL;
	fNewPhi : LREAL;
END_VAR

IF NOT __ISVALIDREF(fbPosition) THEN
	F_RotatePositionXY := E_FAIL;
	RETURN;
END_IF

fRadius := fbPosition.GetRadius();
fPhi := fbPosition.GetPhi();

fNewPhi := MODABS((fPhi + fRotate), 360.0);

fbPosition.SetValuesRP(radius := fRadius, phi := fNewPhi);

END_FUNCTION

// COMPONENTs/Mover/I_XP_Mover
INTERFACE I_XP_Mover  EXTENDS I_CH_Object

PROPERTY DynConstraint : REFERENCE TO DynamicConstraint_Container
GET
END_GET
END_PROPERTY

METHOD SetDynConstraint_A : BOOL //Dynamic constraints for individual coordinates.
VAR_INPUT
    V : MC_LREAL; //equivalent to data type LREAL + MC_DEFAULT, MC_MAXIMUM
    A : MC_LREAL; //equivalent to data type LREAL + MC_DEFAULT, MC_MAXIMUM
    D : MC_LREAL; //equivalent to data type LREAL + MC_DEFAULT, MC_MAXIMUM
    J : MC_LREAL; //equivalent to data type LREAL + MC_DEFAULT, MC_MAXIMUM
END_VAR
END_METHOD

METHOD SetDynConstraint_B : BOOL //Dynamic constraints for individual coordinates.
VAR_INPUT
    V : MC_LREAL; //equivalent to data type LREAL + MC_DEFAULT, MC_MAXIMUM
    A : MC_LREAL; //equivalent to data type LREAL + MC_DEFAULT, MC_MAXIMUM
    D : MC_LREAL; //equivalent to data type LREAL + MC_DEFAULT, MC_MAXIMUM
    J : MC_LREAL; //equivalent to data type LREAL + MC_DEFAULT, MC_MAXIMUM
END_VAR
END_METHOD

METHOD SetDynConstraint_C : BOOL //Dynamic constraints for individual coordinates.
VAR_INPUT
    V : MC_LREAL; //equivalent to data type LREAL + MC_DEFAULT, MC_MAXIMUM
    A : MC_LREAL; //equivalent to data type LREAL + MC_DEFAULT, MC_MAXIMUM
    D : MC_LREAL; //equivalent to data type LREAL + MC_DEFAULT, MC_MAXIMUM
    J : MC_LREAL; //equivalent to data type LREAL + MC_DEFAULT, MC_MAXIMUM
END_VAR
END_METHOD

METHOD SetDynConstraint_Path : BOOL //One dimensional dynamic constraint along the XY-components of a path, ignoring non-tangential effects.
VAR_INPUT
    V : MC_LREAL; //equivalent to data type LREAL + MC_DEFAULT, MC_MAXIMUM
    A : MC_LREAL; //equivalent to data type LREAL + MC_DEFAULT, MC_MAXIMUM
    D : MC_LREAL; //equivalent to data type LREAL + MC_DEFAULT, MC_MAXIMUM
    J : MC_LREAL; //equivalent to data type LREAL + MC_DEFAULT, MC_MAXIMUM
END_VAR
END_METHOD

METHOD SetDynConstraint_X : BOOL //Dynamic constraints for individual coordinates.
VAR_INPUT
    V : MC_LREAL; //equivalent to data type LREAL + MC_DEFAULT, MC_MAXIMUM
    A : MC_LREAL; //equivalent to data type LREAL + MC_DEFAULT, MC_MAXIMUM
    D : MC_LREAL; //equivalent to data type LREAL + MC_DEFAULT, MC_MAXIMUM
    J : MC_LREAL; //equivalent to data type LREAL + MC_DEFAULT, MC_MAXIMUM
END_VAR
END_METHOD

METHOD SetDynConstraint_Y : BOOL //Dynamic constraints for individual coordinates.
VAR_INPUT
    V : MC_LREAL; //equivalent to data type LREAL + MC_DEFAULT, MC_MAXIMUM
    A : MC_LREAL; //equivalent to data type LREAL + MC_DEFAULT, MC_MAXIMUM
    D : MC_LREAL; //equivalent to data type LREAL + MC_DEFAULT, MC_MAXIMUM
    J : MC_LREAL; //equivalent to data type LREAL + MC_DEFAULT, MC_MAXIMUM
END_VAR
END_METHOD

METHOD SetDynConstraint_Z : BOOL //Dynamic constraints for individual coordinates.
VAR_INPUT
    V : MC_LREAL; //equivalent to data type LREAL + MC_DEFAULT, MC_MAXIMUM
    A : MC_LREAL; //equivalent to data type LREAL + MC_DEFAULT, MC_MAXIMUM
    D : MC_LREAL; //equivalent to data type LREAL + MC_DEFAULT, MC_MAXIMUM
    J : MC_LREAL; //equivalent to data type LREAL + MC_DEFAULT, MC_MAXIMUM
END_VAR
END_METHOD

METHOD StopExternalSetpoint : HRESULT
VAR_INPUT
END_VAR
END_METHOD

METHOD AddToGroup : HRESULT
VAR_INPUT
	iGroup : I_XP_Group;
END_VAR
END_METHOD

METHOD RemoveFromGroup : HRESULT
END_METHOD

METHOD Halt : HRESULT
VAR_INPUT
END_VAR
END_METHOD

METHOD MoveA : HRESULT
VAR_INPUT
	fPosition : LREAL;
END_VAR
END_METHOD

METHOD MoveB : HRESULT
VAR_INPUT
	fPosition : LREAL;
END_VAR
END_METHOD

METHOD MoveC : HRESULT
VAR_INPUT
	fPosition : LREAL;
	
	(* Addition turns to move in modulo movement (positive or negative). *)
	additionalTurns : UDINT := 0;
	
	(* Direction in which the target is approached. *)
	direction : Tc3_Mc3Definitions.MC_DIRECTION := Tc3_Mc3Definitions.MC_DIRECTION.mcDirectionNonModulo;
END_VAR
END_METHOD

METHOD MoveXY : HRESULT
VAR_INPUT
	fPosition_X : LREAL;
	fPosition_Y : LREAL;
END_VAR
END_METHOD

METHOD MoveZ : HRESULT
VAR_INPUT
	fPosition : LREAL;
END_VAR
END_METHOD

{attribute 'monitoring':='call'}
(* Velocity is zero *)
PROPERTY Standstill : BOOL
GET
END_GET
END_PROPERTY

METHOD Disable : HRESULT
VAR_INPUT
END_VAR
END_METHOD

METHOD Enable : HRESULT
VAR_INPUT
END_VAR
END_METHOD

METHOD Reset : HRESULT
VAR_INPUT
END_VAR
END_METHOD

{attribute 'monitoring':='call'}
PROPERTY LastCmdTargedGap : LREAL
GET
END_GET
END_PROPERTY

{attribute 'monitoring':='call'}
PROPERTY LastCmdTargedPosition : LREAL
GET
END_GET
END_PROPERTY

{attribute 'monitoring':='call'}
PROPERTY LastCmdTargedTrack: I_XP_Track
GET
END_GET
END_PROPERTY

{attribute 'monitoring':='call'}
//This was the last valid (system enabled) actual  position of the mover
PROPERTY LastValidPositionOnTrack : LREAL
GET
END_GET
END_PROPERTY

{attribute 'monitoring':='call'}
//This was the last valid (system enabled) actual  position of the mover
PROPERTY LastValidPositionXYZABC : REFERENCE TO MoverVector
GET
END_GET
END_PROPERTY

{attribute 'monitoring':='call'}
//This was the last valid (system enabled) actual  position of the mover
PROPERTY LastValidTrack : I_XP_Track;
GET
END_GET
END_PROPERTY

{attribute 'monitoring':='call'}
(* Provides the current planar mover setpoint XYZABC [mm/s²] *)
PROPERTY AccelerationSet : REFERENCE TO MoverVector
GET
END_GET
END_PROPERTY

{attribute 'monitoring':='call'}
(* C coordinate modulus set in MC3-Planar Mover[°] *)
PROPERTY CAxisModulo : LREAL
GET
END_GET
END_PROPERTY

{attribute 'monitoring':='call'}
PROPERTY DistToParentStation : LREAL //Distance to the responsible parent station [mm]
GET
END_GET
END_PROPERTY

{attribute 'monitoring':='call'}
//operational and position control active(hovering)
PROPERTY Enabled : BOOL
GET
END_GET
END_PROPERTY

{attribute 'OPC.UA.DA.Property' := '1'}
{attribute 'monitoring':='call'}
PROPERTY Feedback : I_XP_Feedback
GET
END_GET
END_PROPERTY

{attribute 'monitoring':='call'}
PROPERTY Mapped : BOOL //Project is mapped to MC (McToPlc and PlcToMc)
GET
END_GET
END_PROPERTY

{attribute 'monitoring':='call'}
PROPERTY Mode : MC_PLANAR_MOVER_COMMAND_MODE
GET
END_GET
END_PROPERTY

{attribute 'monitoring':='call'}
(* Height that is used for internal collision checks.[mm] *)
PROPERTY MoverHeight : LREAL
GET
END_GET
END_PROPERTY

{attribute 'monitoring':='call'}
//Mover could not be detected or was removed from the system
PROPERTY MoverIsNotPresent : BOOL
GET
END_GET
END_PROPERTY

{attribute 'monitoring':='call'}
(* Width that is used for internal collision checks.[mm] *)
PROPERTY MoverWidth : LREAL
GET
END_GET
END_PROPERTY

{attribute 'monitoring':='call'}
//Unique object ID
PROPERTY OID : OTCID
GET
END_GET
END_PROPERTY

{attribute 'monitoring':='call'}
(* Provides the current planar mover setpoint XYZABC [mm] *)
PROPERTY PositionSet : REFERENCE TO MoverVector
GET
END_GET
END_PROPERTY

{attribute 'monitoring':='call'}
PROPERTY Route : REFERENCE TO FB_CH_List
GET
END_GET
END_PROPERTY

{attribute 'monitoring':='call'}
(* Provides the current planar mover setpoint XYZABC [mm/s] *)
PROPERTY VelocitySet : REFERENCE TO MoverVector
GET
END_GET
END_PROPERTY

{attribute 'monitoring':='call'}
PROPERTY CurrentTrack : I_XP_Track
GET
END_GET
END_PROPERTY

METHOD DistToTrack : LREAL
VAR_INPUT
	iTrack : I_XP_Track;
END_VAR
END_METHOD

METHOD JoinTrack : HRESULT
VAR_INPUT
	iTrack : I_XP_Track;
END_VAR
END_METHOD

METHOD MoveOnTrack : HRESULT
VAR_INPUT
	ipTrack : I_XP_Track;
	fPosition : LREAL;
	fGap : LREAL;
END_VAR
END_METHOD

METHOD MoveOnTrack_ShortestWay : HRESULT
VAR_INPUT
	ipTrack : I_XP_Track;
	fPosition : LREAL;
	fGap : LREAL;
END_VAR
END_METHOD

METHOD MoveOnTrackToStation : HRESULT
VAR_INPUT
	ipStation : I_XP_Station;
	fGap : LREAL;
END_VAR
END_METHOD

{attribute 'monitoring':='call'}
PROPERTY ParentStation : I_XP_Station
GET
END_GET
SET
END_SET
END_PROPERTY

{attribute 'monitoring':='call'}
PROPERTY PositionOnTrack : Lreal
GET
END_GET
END_PROPERTY

{attribute 'monitoring':='call'}
PROPERTY TargetStation : String
GET
END_GET
SET
END_SET
END_PROPERTY

PROPERTY TcIoXPlanarMover : Tc3_XPlanarUtility.I_TcIoXPlanarMover
GET
END_GET
END_PROPERTY

{attribute 'monitoring':='call'}
PROPERTY UtilityMover : Tc3_XPlanarUtility.I_McPlanarMover
GET
END_GET
END_PROPERTY

{attribute 'monitoring':='call'}
PROPERTY PlanarMover : REFERENCE TO MC_PlanarMover
GET
END_GET
END_PROPERTY

END_INTERFACE

// COMPONENTs/Track/I_XP_Track
INTERFACE I_XP_Track  EXTENDS I_CH_Object

METHOD AddMover : HRESULT
VAR_INPUT
	ipMover : I_XP_Mover;
END_VAR
END_METHOD

METHOD AddToGroup : HRESULT
VAR_INPUT
	iGroup : I_XP_Group;
END_VAR
END_METHOD

{attribute 'monitoring':='call'}
PROPERTY ClosedLoop : BOOL
GET
END_GET
END_PROPERTY

METHOD Configure : HRESULT
VAR_INPUT
END_VAR
END_METHOD

METHOD Configuring : HRESULT
VAR_INPUT
END_VAR
END_METHOD

{attribute 'monitoring':='call'}
PROPERTY CtsMoversOnTrack : UINT
GET
END_GET
END_PROPERTY

METHOD Disable : HRESULT
VAR_INPUT
END_VAR
END_METHOD

METHOD Enable : HRESULT
VAR_INPUT
END_VAR
END_METHOD

{attribute 'monitoring':='call'}
PROPERTY Feedback : I_XP_Feedback
GET
END_GET
END_PROPERTY

(* Calculates which gap the mover should have on a position
	The gap results from the last station crossed.
	If several stations are possible ( switch), the largest gap is displayed here *)
METHOD GapAtPosition : LREAL
VAR_INPUT
	fPosOnTrack : LREAL;//[mm]	
END_VAR
END_METHOD

{attribute 'monitoring':='call'}
//[mm]
PROPERTY Length : LREAL
GET
END_GET
END_PROPERTY

{attribute 'monitoring':='call'}
PROPERTY PlanarTrack : REFERENCE TO MC_PlanarTrack
GET
END_GET
END_PROPERTY

METHOD RemoveFromGroup : HRESULT
END_METHOD

METHOD Reset : HRESULT
VAR_INPUT
END_VAR
END_METHOD

(* Returns the first station on current track who has exact thsi position or is ahead
	If no station on this track, result is maybe on another track*)
METHOD StationAhedPosition : I_XP_Station
VAR_INPUT
	fPosOnTrack : LREAL;//[mm]	
END_VAR
END_METHOD

{attribute 'monitoring':='call'}
//List of interfaces to stations on this track
PROPERTY StationsOnTrack : I_CH_List
GET
END_GET
END_PROPERTY

{attribute 'monitoring':='call'}
//List of interfaces from other tracks
PROPERTY TracksAhead : I_CH_List
GET
END_GET
END_PROPERTY

{attribute 'monitoring':='call'}
//List of interfaces from other tracks
PROPERTY TracksBehinde : I_CH_List
GET
END_GET
END_PROPERTY

{attribute 'monitoring':='call'}
PROPERTY TracksEndAtThis : REFERENCE TO  ARRAY[0..(XPlanarParameterlist.N_MAX_STATIONS_AHEAD_OR_BEHIND-1)] OF I_XP_Track
GET
END_GET
END_PROPERTY

{attribute 'monitoring':='call'}
PROPERTY TracksStartFromThis : REFERENCE TO ARRAY[0..(XPlanarParameterlist.N_MAX_STATIONS_AHEAD_OR_BEHIND-1)] OF I_XP_Track
GET
END_GET
END_PROPERTY

END_INTERFACE

// COMPONENTs/Stationen/I_XP_Station
INTERFACE I_XP_Station EXTENDS I_CH_Object

{attribute 'monitoring':='call'}
//Track on which the station is located
PROPERTY AccocietedTrack : I_XP_Track
GET
END_GET
END_PROPERTY

METHOD AddMoverToQueue : HRESULT
VAR_INPUT
	ipMover : I_XP_Mover;
END_VAR
END_METHOD

{attribute 'monitoring':='call'}
//List of movers managed by this station
PROPERTY AssignedMovers : I_CH_List
GET
END_GET
END_PROPERTY

//Call this Methode whith seq 0->100, and wait each step until S_OK is returned
METHOD Configure : HRESULT
VAR_INPUT
	nSeq : UINT; //0->100
END_VAR
END_METHOD

{attribute 'monitoring':='call'}
PROPERTY CtsEmptySpaceInQueue : UDINT
GET
END_GET
END_PROPERTY

{attribute 'monitoring':='call'}
PROPERTY CtsMoversInQueue : UDINT
GET
END_GET
END_PROPERTY

METHOD DeleteMoversQueue : HRESULT
VAR_INPUT
END_VAR
END_METHOD

{attribute 'monitoring':='call'}
PROPERTY Filter : STRING
GET
END_GET
SET
END_SET
END_PROPERTY

{attribute 'monitoring':='call'}
PROPERTY MoverAccAtExit : MC_LREAL //[mm/s² on Track] Every mover that leaves or passes the station gets this new acceleration as a target.
GET
END_GET
END_PROPERTY

{attribute 'monitoring':='call'}
PROPERTY MoverDecAtExit : MC_LREAL //[mm/s² on Track] Every mover that leaves or passes the station gets this new deceleration as a target.
GET
END_GET
END_PROPERTY

{attribute 'monitoring':='call'}
//[mm] Every mover that leaves or passes the station gets this new gap as a target.
PROPERTY MoverGapAtExit : LREAL
GET
END_GET
SET
END_SET
END_PROPERTY

{attribute 'monitoring':='call'}
PROPERTY MoverQueueSize : UINT
GET
END_GET
END_PROPERTY

{attribute 'monitoring':='call'}
PROPERTY MoversInPlace : BOOL
GET
END_GET
END_PROPERTY

{attribute 'monitoring':='call'}
PROPERTY MoverVelocityAtExit : MC_LREAL //[mm/s on Track] Every mover that leaves or passes the station gets this new velocity as a target.
GET
END_GET
END_PROPERTY

{attribute 'monitoring':='call'}
//List of paths that lead to stations before this station
PROPERTY PathsAhead : I_CH_List
GET
END_GET
END_PROPERTY

{attribute 'monitoring':='call'}
//List of paths that lead to stations behind this station
PROPERTY PathsBehinde : I_CH_List
GET
END_GET
END_PROPERTY

{attribute 'monitoring':='call'}
//[mm] from the beginning of the assigned track
PROPERTY PositionOnTrack : LREAL
GET
END_GET
END_PROPERTY

{attribute 'monitoring':='call'}
//Position on the assigned track
PROPERTY PositionOnTrackXY : REFERENCE TO PositionXY
GET
END_GET
END_PROPERTY

{attribute 'monitoring':='call'}
//Planned position, not necessarily on the track
PROPERTY PositionXY : REFERENCE TO  PositionXY
GET
END_GET
END_PROPERTY

//The movers currently in this station must leave the station. 
//The movers actively search for a destination, but only leave if a new destination is available.
METHOD PushMoversOutOfStation : HRESULT
VAR_INPUT
END_VAR
END_METHOD

{attribute 'monitoring':='call'}
//prevent further movers from entering the station, 
//e.g. to prevent a collision. All movers that are already moving to reach this station will be stopped with a stop 
//and restarted with Ready True.
PROPERTY ReadyToRecvMovers : BOOL
GET
END_GET
END_PROPERTY

METHOD SendMoversToStation : I_CH_Feedback //All movers in the station are sent to this destination
VAR_INPUT
	sTargetStation: STRING;//unique station name or group of stations
END_VAR
END_METHOD

{attribute 'monitoring':='call'}
//List of stations before this station
PROPERTY StationsAhead : I_CH_List
GET
END_GET
END_PROPERTY

{attribute 'monitoring':='call'}
//List of stations behinde this station
PROPERTY StationsBehinde : I_CH_List
GET
END_GET
END_PROPERTY

{attribute 'monitoring':='call'}
PROPERTY TargetGroupe : STRING
GET
END_GET
END_PROPERTY

METHOD Update : HRESULT
VAR_INPUT
END_VAR
END_METHOD

END_INTERFACE

// COMPONENTs/System/I_XP_System_PLC
INTERFACE I_XP_System_PLC EXTENDS I_CH_Object

METHOD CheckTargetExists : BOOL //Return TRUE if target is existing
VAR_INPUT
	sStation	: STRING; //Group of the targed station or LUID
END_VAR
END_METHOD

METHOD Disable : I_CH_Feedback
VAR_INPUT
END_VAR
END_METHOD

{attribute 'monitoring':='call'}
PROPERTY Disabled : BOOL
GET
END_GET
END_PROPERTY

METHOD Enable : I_CH_Feedback
VAR_INPUT
END_VAR
END_METHOD

{attribute 'monitoring':='call'}
PROPERTY Enabled : BOOL
GET
END_GET
END_PROPERTY

{attribute 'monitoring':='call'}
PROPERTY Enviroment : I_XP_Environment
GET
END_GET
END_PROPERTY

METHOD FastStop : I_CH_Feedback
END_METHOD

{attribute 'monitoring':='call'}
PROPERTY Feedback : CHALET_BaseComponents.I_CH_Feedback
GET
END_GET
END_PROPERTY

//Returns the station that is closest to the point according to Phytagoras
METHOD GetStationClosestTo : I_XP_Station
VAR_INPUT
	pos : MoverVector;
END_VAR
END_METHOD

METHOD Initialize : HRESULT
VAR_INPUT
END_VAR
END_METHOD

{attribute 'monitoring':='call'}
PROPERTY Initialized : BOOL
GET
END_GET
END_PROPERTY

{attribute 'monitoring':='call'}
PROPERTY Movers : CHALET_BaseComponents.I_CH_LIST
GET
END_GET
END_PROPERTY

{attribute 'monitoring':='call'}
PROPERTY Paths : CHALET_BaseComponents.I_CH_LIST
GET
END_GET
END_PROPERTY

METHOD Station : I_XP_Station_PLC
VAR_INPUT
	sLUID : STRING;
END_VAR
END_METHOD

{attribute 'monitoring':='call'}
PROPERTY Stations : CHALET_BaseComponents.I_CH_LIST
GET
END_GET
END_PROPERTY

//Suppress to change the dynamic(Gap) of passing movers in all stations. This is usefull in startup
PROPERTY SuppressAllDynamicsChanges : BOOL
SET
END_SET
END_PROPERTY

{attribute 'monitoring':='call'}
PROPERTY Tracks : CHALET_BaseComponents.I_CH_LIST
GET
END_GET
END_PROPERTY

{attribute 'monitoring':='call'}
PROPERTY Triggers : CHALET_BaseComponents.I_CH_LIST
GET
END_GET
END_PROPERTY

METHOD Update : HRESULT
VAR_INPUT
END_VAR
END_METHOD

{attribute 'monitoring':='call'}
PROPERTY Zones : CHALET_BaseComponents.I_CH_LIST
GET
END_GET
END_PROPERTY

END_INTERFACE

// COMPONENTs/Stationen/I_XP_Station_PLC
INTERFACE I_XP_Station_PLC EXTENDS I_CH_Object

{attribute 'monitoring':='call'}
PROPERTY CtsEmptySpaceInQueue : UDINT
GET
END_GET
END_PROPERTY

{attribute 'monitoring':='call'}
PROPERTY CtsMoversInQueue : UDINT
GET
END_GET
END_PROPERTY

{attribute 'monitoring':='call'}
//Filter content, movers with one of these targets may not approach or drive over the station
PROPERTY Filter : STRING
GET
END_GET
SET
END_SET
END_PROPERTY

{attribute 'monitoring':='call'}
PROPERTY LUID : STRING //Locally unique identifier
GET
END_GET
END_PROPERTY

{attribute 'monitoring':='call'}
PROPERTY MoverAccAtExit : MC_LREAL //[mm/s² on Track] Every mover that leaves or passes the station gets this new acceleration as a target.
GET
END_GET
SET
END_SET
END_PROPERTY

{attribute 'monitoring':='call'}
PROPERTY MoverDecAtExit : MC_LREAL //[mm/s² on Track] Every mover that leaves or passes the station gets this new deceleration as a target.
GET
END_GET
SET
END_SET
END_PROPERTY

{attribute 'monitoring':='call'}
PROPERTY MoverQueueSize : UINT
GET
END_GET
SET
END_SET
END_PROPERTY

{attribute 'monitoring':='call'}
PROPERTY MoversInPlace : BOOL
GET
END_GET
END_PROPERTY

{attribute 'monitoring':='call'}
PROPERTY MoversInQueue : REFERENCE TO ARRAY [0..(CHALET_BaseComponents.BaseParameterlist.MAX_OBJECTS-1)] OF I_XP_Mover_PLC // Return a sorted list of movers in this zone. Index 0 is the mover in Front
GET
END_GET
END_PROPERTY

{attribute 'monitoring':='call'}
PROPERTY MoverVelocityAtExit : MC_LREAL //[mm/s on Track] Every mover that leaves or passes the station gets this new velocity as a target.
GET
END_GET
SET
END_SET
END_PROPERTY

//The movers currently in this station must leave the station. 
//The movers actively search for a destination, but only leave if a new destination is available.
METHOD PushMoversOutOfStation : HRESULT
VAR_INPUT
END_VAR
END_METHOD

{attribute 'monitoring':='call'}
//prevent further movers from entering the station, 
//e.g. to prevent a collision. All movers that are already moving to reach this station will be stopped with a stop 
//and restarted with Ready True.
PROPERTY ReadyToRecvMovers : BOOL
GET
END_GET
SET
END_SET
END_PROPERTY

METHOD SendMoversToStation : I_CH_Feedback //All movers in the station are sent to this destination
VAR_INPUT
	sTargetStation: STRING;//unique station name or group of stations
END_VAR
END_METHOD

{attribute 'monitoring':='call'}
//Suppress to change the dynamic(Gap+velocity) of passing movers. This is usefull in startup
PROPERTY SuppressDynamicsChange : BOOL
GET
END_GET
SET
END_SET
END_PROPERTY

{attribute 'monitoring':='call'}
//Interface to CHALET-XPlanar-System
PROPERTY System : I_XP_System_PLC
GET
END_GET
END_PROPERTY

{attribute 'monitoring':='call'}
//A time that is waited as soon as the mover is in the station (including the monitoring window) before “MoversInPlace” is set. e.g. used to stabilize the workpiece
PROPERTY TargetPosMonitoringTime : TIME
GET
END_GET
SET
END_SET
END_PROPERTY

{attribute 'monitoring':='call'}
//How many mm before the mover reaches the position is “MoversInPlace” set for the process. 
//This distance can also be set very large (e.g. 100mm) for moving past without stopping.
PROPERTY TargetPosWindow : LREAL
GET
END_GET
SET
END_SET
END_PROPERTY

{attribute 'monitoring':='call'}
PROPERTY ProcessSimulationActive : BOOL
GET
END_GET
END_PROPERTY

//If a valid time (>0seconds) is set and the configured destination station exists, then the movers will be sent away automatically after this time from now on.
METHOD SimulationStart : HRESULT
VAR_INPUT
	fProcessDuration 		: LREAL; //[s]
	sTargedStation	: STRING; //Group of the targed station to automatic send after the duration
END_VAR
END_METHOD

//If a valid time (>0seconds) is set and the configured destination station exists, then the movers will be sent away automatically after this time from now on.
METHOD SimulationStartEx : HRESULT
VAR_INPUT
	fProcessDuration 		: LREAL; //[s]
	ipStation				: I_XP_Station_PLC; //unique station to automatic send after the duration
END_VAR
END_METHOD

METHOD SimulationStop : HRESULT
END_METHOD

{attribute 'monitoring':='call'}
//Track on which the station is located
PROPERTY AccocietedTrack : I_XP_Track
GET
END_GET
END_PROPERTY

{attribute 'monitoring':='call'}
PROPERTY Feedback : I_CH_Feedback
GET
END_GET
END_PROPERTY

{attribute 'monitoring':='call'}
PROPERTY MoverGapAtExit : LREAL //[mm] Every mover that leaves or passes the station gets this new gap as a target.
GET
END_GET
SET
END_SET
END_PROPERTY

{attribute 'monitoring':='call'}
//[mm] from the beginning of the assigned track
PROPERTY PositionOnTrack : LREAL
GET
END_GET
END_PROPERTY

{attribute 'monitoring':='call'}
//Position on the assigned track
PROPERTY PositionOnTrackXY : REFERENCE TO PositionXY
GET
END_GET
END_PROPERTY

{attribute 'monitoring':='call'}
//Planned position, not necessarily on the track
PROPERTY PositionXY : REFERENCE TO  PositionXY
GET
END_GET
END_PROPERTY

{attribute 'monitoring':='call'}
//List of stations before this station
PROPERTY StationsAhead : I_CH_List
GET
END_GET
END_PROPERTY

{attribute 'monitoring':='call'}
//List of stations behinde this station
PROPERTY StationsBehinde : I_CH_List
GET
END_GET
END_PROPERTY

{attribute 'monitoring':='call'}
PROPERTY TargetGroupe : STRING
GET
END_GET
END_PROPERTY

END_INTERFACE

// COMPONENTs/Mover/I_XP_Mover_PLC
INTERFACE I_XP_Mover_PLC EXTENDS I_CH_Object

PROPERTY DynConstraint : REFERENCE TO DynamicConstraint_Container
GET
END_GET
END_PROPERTY

METHOD SetDynConstraint_A : BOOL //Dynamic constraints for individual coordinates.
VAR_INPUT
    V : MC_LREAL; //equivalent to data type LREAL + MC_DEFAULT, MC_MAXIMUM
    A : MC_LREAL; //equivalent to data type LREAL + MC_DEFAULT, MC_MAXIMUM
    D : MC_LREAL; //equivalent to data type LREAL + MC_DEFAULT, MC_MAXIMUM
    J : MC_LREAL; //equivalent to data type LREAL + MC_DEFAULT, MC_MAXIMUM
END_VAR
END_METHOD

METHOD SetDynConstraint_B : BOOL //Dynamic constraints for individual coordinates.
VAR_INPUT
    V : MC_LREAL; //equivalent to data type LREAL + MC_DEFAULT, MC_MAXIMUM
    A : MC_LREAL; //equivalent to data type LREAL + MC_DEFAULT, MC_MAXIMUM
    D : MC_LREAL; //equivalent to data type LREAL + MC_DEFAULT, MC_MAXIMUM
    J : MC_LREAL; //equivalent to data type LREAL + MC_DEFAULT, MC_MAXIMUM
END_VAR
END_METHOD

METHOD SetDynConstraint_C : BOOL //Dynamic constraints for individual coordinates.
VAR_INPUT
    V : MC_LREAL; //equivalent to data type LREAL + MC_DEFAULT, MC_MAXIMUM
    A : MC_LREAL; //equivalent to data type LREAL + MC_DEFAULT, MC_MAXIMUM
    D : MC_LREAL; //equivalent to data type LREAL + MC_DEFAULT, MC_MAXIMUM
    J : MC_LREAL; //equivalent to data type LREAL + MC_DEFAULT, MC_MAXIMUM
END_VAR
END_METHOD

METHOD SetDynConstraint_Path : BOOL //One dimensional dynamic constraint along the XY-components of a path, ignoring non-tangential effects.
VAR_INPUT
    V : MC_LREAL; //equivalent to data type LREAL + MC_DEFAULT, MC_MAXIMUM
    A : MC_LREAL; //equivalent to data type LREAL + MC_DEFAULT, MC_MAXIMUM
    D : MC_LREAL; //equivalent to data type LREAL + MC_DEFAULT, MC_MAXIMUM
    J : MC_LREAL; //equivalent to data type LREAL + MC_DEFAULT, MC_MAXIMUM
END_VAR
END_METHOD

METHOD SetDynConstraint_X : BOOL //Dynamic constraints for individual coordinates.
VAR_INPUT
    V : MC_LREAL; //equivalent to data type LREAL + MC_DEFAULT, MC_MAXIMUM
    A : MC_LREAL; //equivalent to data type LREAL + MC_DEFAULT, MC_MAXIMUM
    D : MC_LREAL; //equivalent to data type LREAL + MC_DEFAULT, MC_MAXIMUM
    J : MC_LREAL; //equivalent to data type LREAL + MC_DEFAULT, MC_MAXIMUM
END_VAR
END_METHOD

METHOD SetDynConstraint_Y : BOOL //Dynamic constraints for individual coordinates.
VAR_INPUT
    V : MC_LREAL; //equivalent to data type LREAL + MC_DEFAULT, MC_MAXIMUM
    A : MC_LREAL; //equivalent to data type LREAL + MC_DEFAULT, MC_MAXIMUM
    D : MC_LREAL; //equivalent to data type LREAL + MC_DEFAULT, MC_MAXIMUM
    J : MC_LREAL; //equivalent to data type LREAL + MC_DEFAULT, MC_MAXIMUM
END_VAR
END_METHOD

METHOD SetDynConstraint_Z : BOOL //Dynamic constraints for individual coordinates.
VAR_INPUT
    V : MC_LREAL; //equivalent to data type LREAL + MC_DEFAULT, MC_MAXIMUM
    A : MC_LREAL; //equivalent to data type LREAL + MC_DEFAULT, MC_MAXIMUM
    D : MC_LREAL; //equivalent to data type LREAL + MC_DEFAULT, MC_MAXIMUM
    J : MC_LREAL; //equivalent to data type LREAL + MC_DEFAULT, MC_MAXIMUM
END_VAR
END_METHOD

{attribute 'monitoring':='call'}
PROPERTY  AxisExtSetpointA : CHALET_Nc.I_NcAxis_PLC
GET
END_GET
END_PROPERTY

{attribute 'monitoring':='call'}
PROPERTY AxisExtSetpointB : CHALET_Nc.I_NcAxis_PLC
GET
END_GET
END_PROPERTY

{attribute 'monitoring':='call'}
PROPERTY AxisExtSetpointC : CHALET_Nc.I_NcAxis_PLC
GET
END_GET
END_PROPERTY

{attribute 'monitoring':='call'}
PROPERTY  AxisExtSetpointX : CHALET_Nc.I_NcAxis_PLC
GET
END_GET
END_PROPERTY

{attribute 'monitoring':='call'}
PROPERTY AxisExtSetpointY : CHALET_Nc.I_NcAxis_PLC
GET
END_GET
END_PROPERTY

{attribute 'monitoring':='call'}
PROPERTY AxisExtSetpointZ : CHALET_Nc.I_NcAxis_PLC
GET
END_GET
END_PROPERTY

METHOD StartExternalSetpoint : HRESULT
END_METHOD

METHOD StopExternalSetpoint : HRESULT
VAR_INPUT
END_VAR
END_METHOD

METHOD Halt : HRESULT
VAR_INPUT
END_VAR
END_METHOD

METHOD MoveA : HRESULT
VAR_INPUT
	fPosition : LREAL;
END_VAR
END_METHOD

METHOD MoveB : HRESULT
VAR_INPUT
	fPosition : LREAL;
END_VAR
END_METHOD

METHOD MoveC : HRESULT
VAR_INPUT
	fPosition : LREAL;
	
	(* Addition turns to move in modulo movement (positive or negative). *)
	additionalTurns : UDINT := 0;
	
	(* Direction in which the target is approached. *)
	direction : Tc3_Mc3Definitions.MC_DIRECTION := Tc3_Mc3Definitions.MC_DIRECTION.mcDirectionNonModulo;
END_VAR
END_METHOD

METHOD MoveXY : HRESULT
VAR_INPUT
	fPosition_X : LREAL;
	fPosition_Y : LREAL;
END_VAR
END_METHOD

METHOD MoveZ : HRESULT
VAR_INPUT
	fPosition : LREAL;
END_VAR
END_METHOD

{attribute 'monitoring':='call'}
(* Velocity is zero *)
PROPERTY Standstill : BOOL
GET
END_GET
END_PROPERTY

{attribute 'monitoring':='call'}
(* Provides the current planar mover setpoint XYZABC [mm/s²] *)
PROPERTY AccelerationSet : REFERENCE TO MoverVector
GET
END_GET
END_PROPERTY

{attribute 'monitoring':='call'}
(* C coordinate modulus set in MC3-Planar Mover[°] *)
PROPERTY CAxisModulo : LREAL
GET
END_GET
END_PROPERTY

{attribute 'monitoring':='call'}
(* Indicates the command mode of an enabled PlanarMover, i.e. how setpoints are currently produced. *)
PROPERTY CommandMode : MC_PLANAR_MOVER_COMMAND_MODE
GET
END_GET
END_PROPERTY

{attribute 'monitoring':='call'}
//operational and position control active(hovering)
PROPERTY Enabled : BOOL
GET
END_GET
END_PROPERTY

{attribute 'monitoring':='call'}
(* Retruns lentgh of hypotenuse of the x and y error. (>=0[mm]) *)
PROPERTY LagDistanceXY : LREAL
GET
END_GET
END_PROPERTY

{attribute 'monitoring':='call'}
(* Height that is used for internal collision checks.[mm] *)
PROPERTY MoverHeight : LREAL
GET
END_GET
END_PROPERTY

{attribute 'monitoring':='call'}
(* Width that is used for internal collision checks.[mm] *)
PROPERTY MoverWidth : LREAL
GET
END_GET
END_PROPERTY

{attribute 'monitoring':='call'}
(* Contains the information of the Planar Mover passed from MC to PLC. XYZABC [mm] *)
PROPERTY PositionAct : REFERENCE TO MoverVector
GET
END_GET
END_PROPERTY

{attribute 'monitoring':='call'}
(* Provides the current planar mover setpoint XYZABC [mm] *)
PROPERTY PositionSet : REFERENCE TO MoverVector
GET
END_GET
END_PROPERTY

{attribute 'monitoring':='call'}
(* Provides the current planar mover setpoint XYZABC [mm/s] *)
PROPERTY VelocitySet : REFERENCE TO MoverVector
GET
END_GET
END_PROPERTY

{attribute 'monitoring':='call'}
PROPERTY CurrentTrack : I_XP_Track
GET
END_GET
END_PROPERTY

{attribute 'monitoring':='call'}
PROPERTY LastCmdTargedGap : LREAL
GET
END_GET
END_PROPERTY

{attribute 'monitoring':='call'}
PROPERTY LastCmdTargedPosition : LREAL
GET
END_GET
END_PROPERTY

{attribute 'monitoring':='call'}
PROPERTY LastCmdTargedTrack: I_XP_Track
GET
END_GET
END_PROPERTY

METHOD MoveOnTrack : HRESULT
VAR_INPUT
	ipTrack : I_XP_Track;
	fPosition : LREAL;
	fGap : LREAL;
END_VAR
END_METHOD

{attribute 'monitoring':='call'}
PROPERTY ParentStation : I_XP_Station
GET
END_GET
END_PROPERTY

{attribute 'monitoring':='call'}
PROPERTY PositionOnTrack : LREAL
GET
END_GET
END_PROPERTY

{attribute 'monitoring':='call'}
PROPERTY TargetStation : STRING
GET
END_GET
SET
END_SET
END_PROPERTY

{attribute 'monitoring':='call'}
PROPERTY TcIoXPlanarMover : Tc3_XPlanarUtility.I_TcIoXPlanarMover
GET
END_GET
END_PROPERTY

{attribute 'monitoring':='call'}
PROPERTY UtilityMover : Tc3_XPlanarUtility.I_McPlanarMover
GET
END_GET
END_PROPERTY

{attribute 'monitoring':='call'}
PROPERTY DistToParentStation : LREAL //Distance to the responsible parent station [mm]
GET
END_GET
END_PROPERTY

{attribute 'OPC.UA.DA.Property' := '1'}
{attribute 'monitoring':='call'}
PROPERTY Feedback : I_XP_Feedback
GET
END_GET
END_PROPERTY

{attribute 'monitoring':='call'}
PROPERTY LUID : STRING //Locally unique identifier
GET
END_GET
END_PROPERTY

{attribute 'monitoring':='call'}
PROPERTY Mapped : BOOL //Project is mapped to MC (McToPlc and PlcToMc)
GET
END_GET
END_PROPERTY

{attribute 'monitoring':='call'}
//Mover could not be detected or was removed from the system
PROPERTY MoverIsNotPresent : BOOL
GET
END_GET
END_PROPERTY

{attribute 'monitoring':='call'}
//Unique object ID
PROPERTY OID : OTCID
GET
END_GET
END_PROPERTY

{attribute 'monitoring':='call'}
PROPERTY PlanarMover : REFERENCE TO MC_PlanarMover
GET
END_GET
END_PROPERTY

{attribute 'monitoring':='call'}
PROPERTY PUBLIC ProductData : I_XP_ProductData
GET
END_GET
SET
END_SET
END_PROPERTY

END_INTERFACE

// COMPONENTs/Mover/ProductData/I_XP_ProductData
INTERFACE I_XP_ProductData EXTENDS __SYSTEM.IQueryInterface

{attribute 'monitoring':='call'}
PROPERTY LinkedMover : I_XP_Mover_PLC
GET
END_GET
END_PROPERTY

METHOD LinkToMover : BOOL //it is not necessary to call this method. This is already done internally
VAR_INPUT
	ipMoverPlc : I_XP_Mover_PLC;
END_VAR
END_METHOD

END_INTERFACE

// COMPONENTs/Environment/I_XP_Enviroment_PLC
INTERFACE I_XP_Enviroment_PLC EXTENDS I_CH_Object

{attribute 'monitoring':='call'}
(* If Enable, the movers are checked for collisions with each other.
Warning and error can have their own size offsets.
The error leads to a stop with higher dynamics.
In simulation, an error does not lead to a stop *)
PROPERTY CollisionCheck : BOOL
GET
END_GET
SET
END_SET
END_PROPERTY

{attribute 'monitoring':='call'}
//Offset on the mover dimension from the MC3 mover object [mm] ;
// >0 menas the warning is earlier
PROPERTY MoverCollisionOffsetError : LREAL
GET
END_GET
SET
END_SET
END_PROPERTY

{attribute 'monitoring':='call'}
//Offset on the mover dimension from the MC3 mover object [mm] ;
// >0 menas the warning is earlier
PROPERTY MoverCollisionOffsetWarning : LREAL
GET
END_GET
SET
END_SET
END_PROPERTY

{attribute 'monitoring':='call'}
//Enumeration MoverDetectionStatus
PROPERTY MoverDetectionStatus : MoverDetectionStatus
GET
END_GET
END_PROPERTY

{attribute 'monitoring':='call'}
//Object ID of the IoXPlanar processing unit
PROPERTY ProcessingUnitOID : OTCID
GET
END_GET
END_PROPERTY

END_INTERFACE

// COMPONENTs/Group/FB_XP_Group
{attribute 'no_explicit_call' := 'Do not call the body - Stick to OOP'}
(* XPlanar Collision Avoidance Groupe - 1 per associated XPlanar 
	The Planar group is a software object that prevents collisions between Planar movers as well as collisions of Planar movers with the boundary of 
	the stator area on the two-dimensional XPlanar stator area. To do this, the 2D areas of all objects in the group are blocked. When a motion command 
	is transferred to a mover, the required area is requested from the Planar group and the motion command is rejected if this area would collide 
	with already reserved areas. If the motion command can be executed, the area is added to the set of reserved area and blocked accordingly. *)
FUNCTION_BLOCK FB_XP_Group EXTENDS FB_CH_Object IMPLEMENTS I_XP_Group
VAR
	//Link to Planar-Group object
	fbGroup : MC_PlanarGroup;
		
	{attribute 'hide'}  
	bInitDone :BOOL := FALSE;
	{attribute 'hide'}
	iXpSystem : I_XP_System_Registration;
	{attribute 'hide'}               	
	fbFeedback 			: FB_XP_Feedback(ipSourceInfo := fbSourceInfo);	
	{attribute 'hide'}                   	
	eActiveCommand 		: CHALET_Nc.E_NcAxisCommands := CHALET_Nc.E_NcAxisCommands.None;

END_VAR


// Planar-Feedback objects
VAR
	{attribute 'hide'} 
	fbFeedbackDisable : MC_PlanarFeedback;
	{attribute 'hide'} 
	fbFeedbackEnable : MC_PlanarFeedback;
	{attribute 'hide'} 
	fbFeedbackReset : MC_PlanarFeedback;
END_VAR

METHOD AddEnvironment : HRESULT
VAR_INPUT
	refEnvironment : REFERENCE TO MC_PlanarEnvironment;
	refFeedback : REFERENCE TO MC_PlanarFeedback;
END_VAR
refEnvironment.AddToGroup(refFeedback, fbGroup);
END_METHOD

METHOD AddMover : HRESULT
VAR_INPUT
	refMover : REFERENCE TO MC_PlanarMover;
	refFeedback : REFERENCE TO MC_PlanarFeedback;
END_VAR
refMover.AddToGroup(refFeedback, fbGroup);
END_METHOD

METHOD AddTrack : HRESULT
VAR_INPUT
	refTrack : REFERENCE TO MC_PlanarTrack;
	refFeedback : REFERENCE TO MC_PlanarFeedback;
END_VAR
refTrack.AddToGroup(refFeedback, fbGroup);
END_METHOD

METHOD Disable : HRESULT
VAR_INPUT
END_VAR
THIS^.eActiveCommand 				:= CHALET_NC.E_NcAxisCommands.Disable;
THIS^.fbFeedback.LastCommandAccepted:= TRUE;		
THIS^.fbFeedback.Busy 				:= TRUE;

THIS^.fbGroup.Disable(fbFeedbackDisable);

Disable := S_OK;
END_METHOD

METHOD Enable : HRESULT
VAR_INPUT
END_VAR
IF NOT THIS^.fbFeedback.Busy THEN
	THIS^.eActiveCommand 				:= CHALET_NC.E_NcAxisCommands.Enable;
	THIS^.fbFeedback.LastCommandAccepted:= TRUE;		
	THIS^.fbFeedback.Busy 				:= TRUE;

	THIS^.fbGroup.Enable(fbFeedbackEnable);
	Enable := S_OK;
ELSE
	Enable := S_FALSE;
	THIS^.fbFeedback.LastCommandAccepted:= FALSE;	
END_IF
END_METHOD

METHOD FB_init : BOOL
VAR_INPUT
	bInitRetains : BOOL; // if TRUE, the retain variables are initialized (warm start / cold start)
	bInCopyCode : BOOL;  // if TRUE, the instance afterwards gets moved into the copy code (online change)
	
	ipSystem : I_CH_Object;
END_VAR
VAR_INST
	{attribute 'hide'}
	bFBInitCalledOnce : BOOL; //Do the following code once during start up and not during onlinechange
END_VAR
//Do the following code once during start up and not during onlinechange
IF NOT bFBInitCalledOnce THEN 
	

	(* Register to the Xplanar System
	   1. Test if the interface exists
	   2. Test if the object implements a "System for Mover" interface 
	*)
	IF ipSystem <> 0 AND_THEN __QUERYINTERFACE(ipSystem,THIS^.iXpSystem) THEN
		THIS^.iXpSystem.LinkGroup(THIS^);
	END_IF
	
	
END_IF

bFBInitCalledOnce := TRUE;
END_METHOD

{attribute 'monitoring':='call'}
PROPERTY Feedback : I_XP_Feedback
GET
Feedback := THIS^.fbFeedback;
END_GET
END_PROPERTY

METHOD Initialize : HRESULT
VAR_INPUT
END_VAR
VAR
	stVarInfo : __SYSTEM.VAR_INFO;
END_VAR
VAR_INST
	//This error cannot be reset. Requires a reset cold
	{attribute 'hide'}	
	fbInitError : FB_TcAlarm;
END_VAR
// Check if link to MC-Mover is mapped
IF NOT THIS^.Mapped THEN
	IF NOT fbInitError.bRaised THEN 
		//This error cannot be reset. Requires a reset cold
		fbInitError.CreateEx(stEventEntry:=TC_EVENTS.CHALET_Base_Events.VariableLinkMissing, ipSourceInfo := THIS^.fbSourceInfo, bWithConfirmation := FALSE);
		stVarInfo := __VARINFO(fbGroup);
		fbInitError.ipArguments.AddString(stVarInfo.Symbol);
		fbInitError.Raise(0);
	END_IF
	Initialize := E_FAIL;
	RETURN;
END_IF


IF NOT bInitDone THEN
	//Busy
	Initialize := S_PENDING;

	bInitDone := TRUE;	
	
ELSE	
	//Done
	Initialize := S_OK;	
END_IF



THIS^.fbFeedback.ActiveCommand 		:= TO_STRING(CHALET_NC.E_NcAxisCommands.Initialize);
THIS^.eActiveCommand 				:= CHALET_NC.E_NcAxisCommands.Initialize;
THIS^.fbFeedback.LastCommandAccepted:= TRUE;	
//Set done or keep in busy state	
THIS^.fbFeedback.HR := Initialize;
END_METHOD

{attribute 'monitoring':='call'}
PROPERTY Mapped : BOOL //Project is mapped to MC (McToPlc and PlcToMc)
GET
VAR
	bMcToPlcNotMapped 	: BOOL;
END_VAR
bMcToPlcNotMapped := F_GetMappingStatus(ADR(THIS^.fbGroup.MCTOPLC_STD), SIZEOF(THIS^.fbGroup.MCTOPLC_STD)) <> EPlcMappingStatus.MS_Mapped;

Mapped := NOT bMcToPlcNotMapped;
END_GET
END_PROPERTY

{attribute 'monitoring':='call'}
//Unique object ID
PROPERTY OID : OTCID
GET
OID := THIS^.fbGroup.MCTOPLC_STD.GroupOID;
END_GET
END_PROPERTY

{attribute 'monitoring':='call'}
PROPERTY PlanarGroup : REFERENCE TO MC_PlanarGroup
GET
PlanarGroup ref= THIS^.fbGroup;
END_GET
END_PROPERTY

METHOD Reset : HRESULT
VAR_INPUT
END_VAR
IF NOT THIS^.fbFeedback.Busy THEN
	THIS^.eActiveCommand 				:= CHALET_NC.E_NcAxisCommands.Reset;
	THIS^.fbFeedback.LastCommandAccepted:= TRUE;		
	THIS^.fbFeedback.Busy 				:= TRUE;

	THIS^.fbGroup.Reset(fbFeedbackReset);
	Reset := S_OK;
ELSE
	Reset := S_FALSE;
	THIS^.fbFeedback.LastCommandAccepted:= FALSE;		
END_IF
END_METHOD

METHOD PUBLIC Update : HRESULT
VAR_INPUT
END_VAR



// ********************** Set feedback depending on active command *******************************
IF THIS^.eActiveCommand <> E_NcAxisCommands.None THEN
	fbFeedback.ActiveCommand 	:= TO_STRING(THIS^.eActiveCommand);	
END_IF

CASE THIS^.eActiveCommand OF
	E_NcAxisCommands.None: 
		//Display if a Mover Error is active during no command is active
		IF THIS^.fbGroup.Error AND NOT fbFeedback.Error THEN 
			fbFeedback.ErrorId 			:= THIS^.fbGroup.ErrorID;
			fbFeedback.ActiveCommand 	:= TO_STRING(E_NcAxisCommands.None);	
			fbFeedback.ClearObjectInfo();
		END_IF

	E_NcAxisCommands.Initialize:
		fbFeedback.Busy 			:= NOT THIS^.bInitDone;
		fbFeedback.Done 			:= THIS^.bInitDone;
		fbFeedback.ErrorId 			:= 0;
		fbFeedback.ClearObjectInfo();
		                        	
	E_NcAxisCommands.Enable:     	
		fbFeedback.Busy 			:= fbFeedbackEnable.Busy;
		fbFeedback.Done 			:= fbFeedbackEnable.Done;
		fbFeedback.ErrorId 			:= fbFeedbackEnable.ErrorID;
        fbFeedback.ObjectInfo		:= fbFeedbackEnable.objectInfo;
                                			                        	
	E_NcAxisCommands.Disable:     	
		fbFeedback.Busy 			:= fbFeedbackDisable.Busy;
		fbFeedback.Done 			:= fbFeedbackDisable.Done;
		fbFeedback.ErrorId 			:= fbFeedbackDisable.ErrorID;
        fbFeedback.ObjectInfo		:= fbFeedbackDisable.objectInfo;
                                			                        	
	E_NcAxisCommands.Reset:     	
		fbFeedback.Busy 			:= fbFeedbackReset.Busy;
		fbFeedback.Done 			:= fbFeedbackReset.Done;
		fbFeedback.ErrorId 			:= fbFeedbackReset.ErrorID;
        fbFeedback.ObjectInfo		:= fbFeedbackReset.objectInfo;
                                		
	ELSE//External command in subclass
		;
END_CASE


// **********************  Stop to execute commands on .done or .error ***************************
IF fbFeedback.Done OR THIS^.fbFeedback.Error THEN
	eActiveCommand 				:= E_NcAxisCommands.None;
END_IF

//Update xplanar object
THIS^.fbGroup.Update();

//Update feedback object
fbFeedbackEnable.Update(); 
fbFeedbackDisable.Update(); 
fbFeedbackReset.Update();
END_METHOD

END_FUNCTION_BLOCK

// COMPONENTs/Mover/ProductData/FB_XP_ProductData
FUNCTION_BLOCK FB_XP_ProductData EXTENDS FB_CH_Object IMPLEMENTS I_XP_ProductData
VAR
	{attribute 'hide'}
	ipMover : I_XP_Mover_PLC;
END_VAR

{attribute 'monitoring':='call'}
PROPERTY LinkedMover : I_XP_Mover_PLC
GET
LinkedMover := ipMover;
END_GET
END_PROPERTY

METHOD LinkToMover : BOOL //it is not necessary to call this method. This is already done internally
VAR_INPUT
	ipMoverPlc : I_XP_Mover_PLC;
END_VAR
THIS^.ipMover := ipMoverPlc;
END_METHOD

END_FUNCTION_BLOCK

// COMPONENTs/Mover/FB_XP_Mover
// The warning " Interface of overridden methode xxx of base I_xxx doesn't match declaration" can be disabled here. 
{warning disable C0094 }
{attribute 'no_explicit_call' := 'Do not call the body - Stick to OOP'}
(* XPlanar mover - n per associated XPlanar. Can be instantiated as an array and/or individually
	The Planar mover is a software object that represents an XPlanar mover. It summarizes the state of the real mover (position, velocity, etc.) 
	for the user. In addition, the user has the possibility to influence or control the state of the real mover via the Planar mover. *)	
FUNCTION_BLOCK FB_XP_Mover EXTENDS FB_CH_Object IMPLEMENTS I_XP_Mover, I_XP_Mover_PLC
VAR
	fbRoute : FB_CH_List;
END_VAR

VAR
	//Link to MC-Mover
	fbMover : MC_PlanarMover;
	
	{attribute 'hide'}  
	bInitDone :BOOL := FALSE;
	{attribute 'hide'}               	
	fbFeedback 			: FB_XP_Feedback(ipSourceInfo := fbSourceInfo);	
	{attribute 'hide'}                   	
	eActiveCommand 		: CHALET_Nc.E_NcAxisCommands := CHALET_Nc.E_NcAxisCommands.None;
	{attribute 'hide'} 
	fbUtilityMover : FB_McPlanarMover;
	{attribute 'hide'}
	ipXpSystem : I_XP_System_Registration;
	{attribute 'hide'} 
	sTargedStation : STRING := XPlanarParameterlist.S_MOVER_TARGED_INIT;
	{attribute 'hide'} 
	sCurrentStation : STRING;
	{attribute 'hide'}
	ipParentStation : I_XP_Station; //This is the station in which the Mover is currently standing or moving.	
	{attribute 'hide'}
	ipProductData : I_XP_ProductData; //later the required interface of the tool or product can be queried via query interface
END_VAR

//Recovery
VAR
	{attribute 'hide'}
	//This was the last valid (system enabled) actual  position of the mover
	stLastValidPositionXYZABC :  MoverVector;
	{attribute 'hide'}
	//This was the last valid (system enabled) actual  position of the mover
	fLastValidPositionOnTrack :  LREAL;
	{attribute 'hide'}
	//This was the last valid (system enabled) actual  position of the mover
	ipLastValidTrack : I_XP_Track;
	{attribute 'hide'}
	fLastCmdTargedPosition : LREAL; //the last commanded target position [mm]
	{attribute 'hide'}	
	fLastCmdTargedGap 	: LREAL; //the last commanded target gap
	{attribute 'hide'}		
	ipLastCmdTrack : I_XP_Track;	
END_VAR


//External Setpoint Generator
VAR
	AxisSetpointX : FB_NcAxis;
	AxisSetpointY : FB_NcAxis;
	AxisSetpointZ : FB_NcAxis;
	AxisSetpointA : FB_NcAxis;
	AxisSetpointB : FB_NcAxis;
	AxisSetpointC : FB_NcAxis;
//	{attribute 'hide'} 
	nSeqStartExternalSetpoint : UINT;
//	{attribute 'hide'} 	
	//As long as the bit is still false, the MC_PlanarFeedback should not be evaluated as it may still indicate an old error
	bEvaluateFeedback: BOOL; 
//	{attribute 'hide'} 
	bFeedExternalSetpointActive : BOOL; 
//	{attribute 'hide'} 
	fbFeedbackExternalSetpointStartSeq : FB_CH_Feedback(0);
//	{attribute 'hide'} 
	ipMasterMover : I_XP_Mover;

	
//	{attribute 'hide'} 
	stMasterMovementScaling : MoverVector; // if 0, Mover is not folowing this mover axis
//	{attribute 'hide'} 
	stMasterPositionAtStart : MoverVector;
	
	
	
END_VAR


//DynamicConstraint
VAR
	{attribute 'hide'} 
	fbDynConstraintContainer 	: DynamicConstraint_Container;		//A container for dynamic constraints.
	{attribute 'hide'} 
	fbDynConstraintPath 		: DynamicConstraint_PathXY; 		//One dimensional dynamic constraint along the XY-components of a path, ignoring non-tangential effects.
	{attribute 'hide'} 	
	fbDynConstraintCoordinates	: DynamicConstraint_Coordinates;	//Dynamic constraints for individual coordinates.
END_VAR


// Planar-Feedback objects
VAR
	{attribute 'hide'} 
	fbFeedbackMoveA : MC_PlanarFeedback;
	{attribute 'hide'} 
	fbFeedbackMoveB : MC_PlanarFeedback;
	{attribute 'hide'} 
	fbFeedbackMoveC : MC_PlanarFeedback;
	{attribute 'hide'} 
	fbFeedbackMoveXY : MC_PlanarFeedback;
	{attribute 'hide'} 
	fbFeedbackMoveZ : MC_PlanarFeedback;
	{attribute 'hide'} 
	fbFeedbackEnable : MC_PlanarFeedback;
	{attribute 'hide'} 
	fbFeedbackDisable : MC_PlanarFeedback;
	{attribute 'hide'} 
	fbFeedbackHalt : MC_PlanarFeedback;
	{attribute 'hide'} 
	fbFeedbackReset : MC_PlanarFeedback;
	{attribute 'hide'} 
	fbFeedbackAddToGrp : MC_PlanarFeedback;
	{attribute 'hide'} 
	fbFeedbackRmvFromGrp : MC_PlanarFeedback;
	{attribute 'hide'} 
	fbFeedbackJoinTrack : MC_PlanarFeedback;
	{attribute 'hide'} 
	fbFeedbackMoveOnTrack: MC_PlanarFeedback;	
	{attribute 'hide'} 
	fbFeedbackExtStart : MC_PlanarFeedback;
	{attribute 'hide'} 
	fbFeedbackExtStop : MC_PlanarFeedback;
END_VAR
{warning restore C0094}

PROPERTY DynConstraint : REFERENCE TO DynamicConstraint_Container
GET
DynConstraint REF= THIS^.fbDynConstraintContainer;
END_GET
END_PROPERTY

METHOD SetDynConstraint_A : BOOL //Dynamic constraints for individual coordinates.
VAR_INPUT
    V : MC_LREAL; //equivalent to data type LREAL + MC_DEFAULT, MC_MAXIMUM
    A : MC_LREAL; //equivalent to data type LREAL + MC_DEFAULT, MC_MAXIMUM
    D : MC_LREAL; //equivalent to data type LREAL + MC_DEFAULT, MC_MAXIMUM
    J : MC_LREAL; //equivalent to data type LREAL + MC_DEFAULT, MC_MAXIMUM
END_VAR
THIS^.fbDynConstraintCoordinates.SetLimit(	Coordinate := Coord_Mcs_A1, 
											V := V, 
											A := A, 
											D := D, 
											J := J);
											
//Changes to the origin constraint do not affect the copy of the constraint in the instance of the DynamicConstraint_Container.
//For this reason, the container is being refreshed here							
fbDynConstraintContainer.Clear();
fbDynConstraintContainer.AddConstraint(fbDynConstraintPath);
fbDynConstraintContainer.AddConstraint(fbDynConstraintCoordinates);
END_METHOD

METHOD SetDynConstraint_B : BOOL //Dynamic constraints for individual coordinates.
VAR_INPUT
    V : MC_LREAL; //equivalent to data type LREAL + MC_DEFAULT, MC_MAXIMUM
    A : MC_LREAL; //equivalent to data type LREAL + MC_DEFAULT, MC_MAXIMUM
    D : MC_LREAL; //equivalent to data type LREAL + MC_DEFAULT, MC_MAXIMUM
    J : MC_LREAL; //equivalent to data type LREAL + MC_DEFAULT, MC_MAXIMUM
END_VAR
THIS^.fbDynConstraintCoordinates.SetLimit(	Coordinate := Coord_Mcs_B1, 
											V := V, 
											A := A, 
											D := D, 
											J := J);											

//Changes to the origin constraint do not affect the copy of the constraint in the instance of the DynamicConstraint_Container.
//For this reason, the container is being refreshed here							
fbDynConstraintContainer.Clear();
fbDynConstraintContainer.AddConstraint(fbDynConstraintPath);
fbDynConstraintContainer.AddConstraint(fbDynConstraintCoordinates);
END_METHOD

METHOD SetDynConstraint_C : BOOL //Dynamic constraints for individual coordinates.
VAR_INPUT
    V : MC_LREAL; //equivalent to data type LREAL + MC_DEFAULT, MC_MAXIMUM
    A : MC_LREAL; //equivalent to data type LREAL + MC_DEFAULT, MC_MAXIMUM
    D : MC_LREAL; //equivalent to data type LREAL + MC_DEFAULT, MC_MAXIMUM
    J : MC_LREAL; //equivalent to data type LREAL + MC_DEFAULT, MC_MAXIMUM
END_VAR
THIS^.fbDynConstraintCoordinates.SetLimit(	Coordinate := Coord_Mcs_C1, 
											V := V, 
											A := A, 
											D := D, 
											J := J);											

//Changes to the origin constraint do not affect the copy of the constraint in the instance of the DynamicConstraint_Container.
//For this reason, the container is being refreshed here							
fbDynConstraintContainer.Clear();
fbDynConstraintContainer.AddConstraint(fbDynConstraintPath);
fbDynConstraintContainer.AddConstraint(fbDynConstraintCoordinates);
END_METHOD

METHOD SetDynConstraint_Path : BOOL //One dimensional dynamic constraint along the XY-components of a path, ignoring non-tangential effects.
VAR_INPUT
    V : MC_LREAL; //equivalent to data type LREAL + MC_DEFAULT, MC_MAXIMUM
    A : MC_LREAL; //equivalent to data type LREAL + MC_DEFAULT, MC_MAXIMUM
    D : MC_LREAL; //equivalent to data type LREAL + MC_DEFAULT, MC_MAXIMUM
    J : MC_LREAL; //equivalent to data type LREAL + MC_DEFAULT, MC_MAXIMUM
END_VAR
THIS^.fbDynConstraintPath.SetValuesVADJ(V := V, 
										A := A, 
										D := D, 
										J := J);											

//Changes to the origin constraint do not affect the copy of the constraint in the instance of the DynamicConstraint_Container.
//For this reason, the container is being refreshed here							
fbDynConstraintContainer.Clear();
fbDynConstraintContainer.AddConstraint(fbDynConstraintPath);
fbDynConstraintContainer.AddConstraint(fbDynConstraintCoordinates);
END_METHOD

METHOD SetDynConstraint_X : BOOL //Dynamic constraints for individual coordinates.
VAR_INPUT
    V : MC_LREAL; //equivalent to data type LREAL + MC_DEFAULT, MC_MAXIMUM
    A : MC_LREAL; //equivalent to data type LREAL + MC_DEFAULT, MC_MAXIMUM
    D : MC_LREAL; //equivalent to data type LREAL + MC_DEFAULT, MC_MAXIMUM
    J : MC_LREAL; //equivalent to data type LREAL + MC_DEFAULT, MC_MAXIMUM
END_VAR
THIS^.fbDynConstraintCoordinates.SetLimit(	Coordinate := Coord_Mcs_X, 
											V := V, 
											A := A, 
											D := D, 
											J := J);											

//Changes to the origin constraint do not affect the copy of the constraint in the instance of the DynamicConstraint_Container.
//For this reason, the container is being refreshed here							
fbDynConstraintContainer.Clear();
fbDynConstraintContainer.AddConstraint(fbDynConstraintPath);
fbDynConstraintContainer.AddConstraint(fbDynConstraintCoordinates);
END_METHOD

METHOD SetDynConstraint_Y : BOOL //Dynamic constraints for individual coordinates.
VAR_INPUT
    V : MC_LREAL; //equivalent to data type LREAL + MC_DEFAULT, MC_MAXIMUM
    A : MC_LREAL; //equivalent to data type LREAL + MC_DEFAULT, MC_MAXIMUM
    D : MC_LREAL; //equivalent to data type LREAL + MC_DEFAULT, MC_MAXIMUM
    J : MC_LREAL; //equivalent to data type LREAL + MC_DEFAULT, MC_MAXIMUM
END_VAR
THIS^.fbDynConstraintCoordinates.SetLimit(	Coordinate := Coord_Mcs_Y, 
											V := V, 
											A := A, 
											D := D, 
											J := J);											

//Changes to the origin constraint do not affect the copy of the constraint in the instance of the DynamicConstraint_Container.
//For this reason, the container is being refreshed here							
fbDynConstraintContainer.Clear();
fbDynConstraintContainer.AddConstraint(fbDynConstraintPath);
fbDynConstraintContainer.AddConstraint(fbDynConstraintCoordinates);
END_METHOD

METHOD SetDynConstraint_Z : BOOL //Dynamic constraints for individual coordinates.
VAR_INPUT
    V : MC_LREAL; //equivalent to data type LREAL + MC_DEFAULT, MC_MAXIMUM
    A : MC_LREAL; //equivalent to data type LREAL + MC_DEFAULT, MC_MAXIMUM
    D : MC_LREAL; //equivalent to data type LREAL + MC_DEFAULT, MC_MAXIMUM
    J : MC_LREAL; //equivalent to data type LREAL + MC_DEFAULT, MC_MAXIMUM
END_VAR
THIS^.fbDynConstraintCoordinates.SetLimit(	Coordinate := Coord_Mcs_Z, 
											V := MC_DEFAULT, 
											A := A, 
											D := D, 
											J := J);											

//Changes to the origin constraint do not affect the copy of the constraint in the instance of the DynamicConstraint_Container.
//For this reason, the container is being refreshed here							
fbDynConstraintContainer.Clear();
fbDynConstraintContainer.AddConstraint(fbDynConstraintPath);
fbDynConstraintContainer.AddConstraint(fbDynConstraintCoordinates);
END_METHOD

//Save the master mover and apply the distance traveled as a relative offset to this slave mover. Requires .StartExternalSetpoint()
METHOD AddMoverExtSetpoint : HRESULT
VAR_INPUT
	ipMasterMover : I_XP_Mover;
	fScalingX, fScalingY, fScalingZ, fScalingA, fScalingB, fScalingC : LREAL;// If >0, follow this axis to master-mover
END_VAR
//Invalide input
IF ipMasterMover = 0 THEN
	AddMoverExtSetpoint := E_FAIL;
	RETURN;
END_IF

//Allready stored a master
IF THIS^.ipMasterMover <> 0 THEN
	AddMoverExtSetpoint := E_FAIL;
	RETURN;
END_IF

//Only possible if ExternalSetpoint is not running
IF THIS^.nSeqStartExternalSetpoint <> 0 THEN
	AddMoverExtSetpoint := E_FAIL;
	RETURN;
END_IF



THIS^.ipMasterMover := ipMasterMover;
THIS^.stMasterMovementScaling.x := fScalingX;
THIS^.stMasterMovementScaling.y := fScalingy;
THIS^.stMasterMovementScaling.z := fScalingz;
THIS^.stMasterMovementScaling.a := fScalinga;
THIS^.stMasterMovementScaling.b := fScalingb;
THIS^.stMasterMovementScaling.c := fScalingc;
END_METHOD

{attribute 'monitoring':='call'}
PROPERTY  AxisExtSetpointA : CHALET_Nc.I_NcAxis_PLC
GET
AxisExtSetpointA := THIS^.AxisSetpointA;
END_GET
END_PROPERTY

{attribute 'monitoring':='call'}
PROPERTY AxisExtSetpointB : CHALET_Nc.I_NcAxis_PLC
GET
AxisExtSetpointB := THIS^.AxisSetpointB;
END_GET
END_PROPERTY

{attribute 'monitoring':='call'}
PROPERTY AxisExtSetpointC : CHALET_Nc.I_NcAxis_PLC
GET
AxisExtSetpointC := THIS^.AxisSetpointC;
END_GET
END_PROPERTY

{attribute 'monitoring':='call'}
PROPERTY  AxisExtSetpointX : CHALET_Nc.I_NcAxis_PLC
GET
AxisExtSetpointX := THIS^.AxisSetpointX;
END_GET
END_PROPERTY

{attribute 'monitoring':='call'}
PROPERTY AxisExtSetpointY : CHALET_Nc.I_NcAxis_PLC
GET
AxisExtSetpointY := THIS^.AxisSetpointY;
END_GET
END_PROPERTY

{attribute 'monitoring':='call'}
PROPERTY AxisExtSetpointZ : CHALET_Nc.I_NcAxis_PLC
GET
AxisExtSetpointZ := THIS^.AxisSetpointZ;
END_GET
END_PROPERTY

METHOD StartExternalSetpoint : HRESULT
THIS^.eActiveCommand 				:= CHALET_NC.E_NcAxisCommands.StartExternalSetpoint;
THIS^.fbFeedback.ActiveCommand 		:= TO_STRING(THIS^.eActiveCommand);		
THIS^.fbFeedback.Busy 				:= TRUE;


IF THIS^.fbMover.MCTOPLC.STD.State <> MC_PLANAR_STATE.Enabled THEN
	//Error wrong state
	
	;//zzz Todo Error message

ELSIF THIS^.bFeedExternalSetpointActive AND THIS^.nSeqStartExternalSetpoint = 999 THEN
	//Do nothing, setpoint is already active	
	THIS^.fbFeedbackExternalSetpointStartSeq.Done		:= TRUE;
	
ELSE
	
	//Start of internal sequence
	THIS^.fbFeedbackExternalSetpointStartSeq.Busy		:= TRUE;
	THIS^.nSeqStartExternalSetpoint := 1;
END_IF



StartExternalSetpoint := S_OK;
END_METHOD

METHOD StopExternalSetpoint : HRESULT
VAR_INPUT
END_VAR
AxisSetpointX.PowerOff();
AxisSetpointY.PowerOff();
AxisSetpointZ.PowerOff();
AxisSetpointA.PowerOff();
AxisSetpointB.PowerOff();
AxisSetpointC.PowerOff();


THIS^.eActiveCommand 				:= CHALET_NC.E_NcAxisCommands.StopExternalSetpoint;
THIS^.fbFeedback.ActiveCommand 		:= TO_STRING(THIS^.eActiveCommand);	
THIS^.fbFeedback.LastCommandAccepted:= TRUE;		


//Reset some flags
THIS^.nSeqStartExternalSetpoint := 0;
THIS^.bEvaluateFeedback := FALSE;
THIS^.ipMasterMover := 0;

IF THIS^.bFeedExternalSetpointActive THEN
	THIS^.fbMover.StopExternalSetpointGeneration(THIS^.fbFeedbackExtStop);	
	THIS^.bFeedExternalSetpointActive 	:= FALSE;
	THIS^.fbFeedback.Busy 				:= TRUE;
ELSE
	THIS^.fbFeedback.Done 				:= TRUE;
END_IF


StopExternalSetpoint := S_OK;
END_METHOD

METHOD PROTECTED UpdateExternalSetpoint : HRESULT
VAR
	SetPos, SetVelo, SetAcc : MoverVector;
	hr : HRESULT;
	stStartOptions : ST_ExternalSetpointGenerationOptions;
	stPosDifferenceToMasterMover : MoverVector;
	stPosOffsetMasterMover : MoverVector;
	stVeloOffsetMasterMover : MoverVector;
	stAccOffsetMasterMover : MoverVector;
END_VAR
IF NOT THIS^.Enabled THEN
	THIS^.nSeqStartExternalSetpoint := 0;
	THIS^.bFeedExternalSetpointActive := FALSE;
	THIS^.bEvaluateFeedback := FALSE;
END_IF


CASE nSeqStartExternalSetpoint OF
	0: //Wait for start
		;
		
	1: 	//store position of Master-Mover
		IF (THIS^.ipMasterMover <> 0) THEN
			THIS^.stMasterPositionAtStart := THIS^.ipMasterMover.PositionSet;
		END_IF

		//Reset all axis
		IF AxisSetpointX.Mapped THEN
			AxisSetpointX.Reset();
		END_IF
		IF AxisSetpointY.Mapped THEN
			AxisSetpointY.Reset();
		END_IF
		IF AxisSetpointZ.Mapped THEN
			AxisSetpointZ.Reset();
		END_IF
		IF AxisSetpointA.Mapped THEN
			AxisSetpointA.Reset();
		END_IF
		IF AxisSetpointB.Mapped THEN
			AxisSetpointB.Reset();
		END_IF
		IF AxisSetpointC.Mapped THEN
			AxisSetpointC.Reset();
		END_IF
		nSeqStartExternalSetpoint := nSeqStartExternalSetpoint + 1;		
		
		
	2: //Wait for feedback
		IF AxisSetpointX.Mapped THEN hr := GetMostSignificant(hr, AxisSetpointX.Feedback.HR); END_IF
		IF AxisSetpointY.Mapped THEN hr := GetMostSignificant(hr, AxisSetpointY.Feedback.HR); END_IF
		IF AxisSetpointZ.Mapped THEN hr := GetMostSignificant(hr, AxisSetpointZ.Feedback.HR); END_IF
		IF AxisSetpointA.Mapped THEN hr := GetMostSignificant(hr, AxisSetpointA.Feedback.HR); END_IF
		IF AxisSetpointB.Mapped THEN hr := GetMostSignificant(hr, AxisSetpointB.Feedback.HR); END_IF
		IF AxisSetpointC.Mapped THEN hr := GetMostSignificant(hr, AxisSetpointC.Feedback.HR); END_IF	
		IF hr = S_OK THEN
		 	nSeqStartExternalSetpoint := nSeqStartExternalSetpoint + 1;	
		END_IF
		
	3: 	//Reset all axis
		IF AxisSetpointX.Mapped THEN
			AxisSetpointX.PowerOn();
		END_IF
		IF AxisSetpointY.Mapped THEN
			AxisSetpointY.PowerOn();
		END_IF
		IF AxisSetpointZ.Mapped THEN
			AxisSetpointZ.PowerOn();
		END_IF
		IF AxisSetpointA.Mapped THEN
			AxisSetpointA.PowerOn();
		END_IF
		IF AxisSetpointB.Mapped THEN
			AxisSetpointB.PowerOn();
		END_IF
		IF AxisSetpointC.Mapped THEN
			AxisSetpointC.PowerOn();
		END_IF
		nSeqStartExternalSetpoint := nSeqStartExternalSetpoint + 1;		
		
	4: //Wait for feedback
		IF AxisSetpointX.Mapped THEN hr := GetMostSignificant(hr, AxisSetpointX.Feedback.HR); END_IF
		IF AxisSetpointY.Mapped THEN hr := GetMostSignificant(hr, AxisSetpointY.Feedback.HR); END_IF
		IF AxisSetpointZ.Mapped THEN hr := GetMostSignificant(hr, AxisSetpointZ.Feedback.HR); END_IF
		IF AxisSetpointA.Mapped THEN hr := GetMostSignificant(hr, AxisSetpointA.Feedback.HR); END_IF
		IF AxisSetpointB.Mapped THEN hr := GetMostSignificant(hr, AxisSetpointB.Feedback.HR); END_IF
		IF AxisSetpointC.Mapped THEN hr := GetMostSignificant(hr, AxisSetpointC.Feedback.HR); END_IF	
		IF hr = S_OK THEN
		 	nSeqStartExternalSetpoint := nSeqStartExternalSetpoint + 1;	
		END_IF

	5: 	//Enable all axis
		IF AxisSetpointX.Mapped THEN
			AxisSetpointX.SetActPosition(0.0);
		END_IF
		IF AxisSetpointY.Mapped THEN
			AxisSetpointY.SetActPosition(0.0);
		END_IF
		IF AxisSetpointZ.Mapped THEN
			AxisSetpointZ.SetActPosition(0.0);
		END_IF
		IF AxisSetpointA.Mapped THEN
			AxisSetpointA.SetActPosition(0.0);
		END_IF
		IF AxisSetpointB.Mapped THEN
			AxisSetpointB.SetActPosition(0.0);
		END_IF
		IF AxisSetpointC.Mapped THEN
			AxisSetpointC.SetActPosition(0.0);
		END_IF
		nSeqStartExternalSetpoint := nSeqStartExternalSetpoint + 1;		
		
	6: //Wait for feedback
		IF AxisSetpointX.Mapped THEN hr := GetMostSignificant(hr, AxisSetpointX.Feedback.HR); END_IF
		IF AxisSetpointY.Mapped THEN hr := GetMostSignificant(hr, AxisSetpointY.Feedback.HR); END_IF
		IF AxisSetpointZ.Mapped THEN hr := GetMostSignificant(hr, AxisSetpointZ.Feedback.HR); END_IF
		IF AxisSetpointA.Mapped THEN hr := GetMostSignificant(hr, AxisSetpointA.Feedback.HR); END_IF
		IF AxisSetpointB.Mapped THEN hr := GetMostSignificant(hr, AxisSetpointB.Feedback.HR); END_IF
		IF AxisSetpointC.Mapped THEN hr := GetMostSignificant(hr, AxisSetpointC.Feedback.HR); END_IF	
		IF hr = S_OK THEN
		 	nSeqStartExternalSetpoint := nSeqStartExternalSetpoint + 1;	
		END_IF

		
